(* POU FB_BACnet_RemoteAccumulator_EX, ST *)
FUNCTION_BLOCK FB_BACnet_RemoteAccumulator_EX
VAR_IN_OUT
	RemoteDevice		: FB_BACnet_RemoteDevice;
END_VAR
VAR_OUTPUT
	bReady				: BOOL;
	nPresentValue		: UDINT;
	bOverridden			: BOOL;
	bOutOfService		: BOOL;
	bFault				: BOOL;
	bInAlarm			: BOOL;
	bOverRange			: BOOL;
	bUnderRange			: BOOL;
	bNoSensor			: BOOL;
	bOpenLoop			: BOOL;
	bCommFailure		: BOOL;
	bShortedLoop		: BOOL;
	bOtherFault			: BOOL;
	tObjectID			: T_BACnet_ObjectIdentifier := 16#FFFFFFFF;
	bError				: BOOL;
	nErrorId			: UINT;
END_VAR
VAR
	_PresentValue AT%I*:UDINT;			(* ~(BACnet_PresentValue				:		: )
											(BACnet_ObjectType					: ACC	: )
											(BACnet_RemoteCycletimeRead			: 1000	: )
											(BACnet_RemoteFlagsRead				: 1		: )
											(BACnet_RemoteResubscriptionInterval: 240	: )
                                			(BACnet_RemoteCycleTimeWrite   		: 1000	: )
                                			(BACnet_RemoteFlagsWrite       		: 1		: )	*)
	_ObjectId AT%I*: DWORD;				(* ~(BACnet_ObjectIdentifier			:		: LINK) *)
	_StatusFlags AT%I*:WORD;			(* ~(BACnet_StatusFlags					:		: )	*)
	_Reliability AT%I*:WORD;			(* ~(BACnet_Reliability					:		: )	*)
	_StatusFlagsBits : ST_BACnet_StatusFlags;

	_nUpdateCount : UDINT := 0;
END_VAR
(* update client device *)
IF RemoteDevice._nUpdateCount = _nUpdateCount THEN
	RemoteDevice();
END_IF
(* remind current number of update counter *)
_nUpdateCount := RemoteDevice._nUpdateCount;

IF NOT RemoteDevice.bOperational THEN
	nErrorId := BACnet_ERR_OPERATIONAL;
	bReady := FALSE;

ELSIF (F_BACnet_GetObjType(_ObjectId) <> BACnetObjectType_Accumulator) THEN
	(* wrong mapping / invalid object ID *)
	IF _ObjectId = 0 THEN
		nErrorId := BACnet_ERR_WRONG_MAPPING;
	ELSE
		nErrorId := BACnet_ERR_INVALID_OBJECTID;
	END_IF
	bReady := FALSE;
	tObjectID := 16#FFFFFFFF;

ELSIF _StatusFlags >= 4 THEN
	(* clear error flag *)
	nErrorId := BACnet_ERR_NO_ERROR;
	bReady := TRUE;
	(* copy present value *)
	nPresentValue := _PresentValue;

	(* build bit states *)
	_StatusFlagsBits := F_BACnet_StatusFlags(_StatusFlags);

	(* copy states to output *)
	bOverridden := _StatusFlagsBits.overridden;
	bOutOfService := _StatusFlagsBits.out_of_service;
	bFault := _StatusFlagsBits.fault;
	bInAlarm := _StatusFlagsBits.in_alarm;
	bOverRange := (_Reliability = BACnetReliability_over_range);
	bUnderRange := (_Reliability = BACnetReliability_under_range);
	bNoSensor := (_Reliability = BACnetReliability_no_sensor);
	bOpenLoop := (_Reliability = BACnetReliability_open_loop);
	bCommFailure := (_Reliability = BACnetReliability_communication_failure);
	bShortedLoop := (_Reliability = BACnetReliability_shorted_loop);
	bOtherFault := (_Reliability = BACnetReliability_unreliable_other);
	tObjectID := _ObjectId;

ELSE
	bReady := FALSE;
	(* and set error ID *)
	nErrorId := BACnet_ERR_WRONG_MAPPING;
END_IF

(* set error flag *)
bError := (nErrorId <> BACnet_ERR_NO_ERROR);
END_FUNCTION_BLOCK

(* POU FB_BACnet_RemoteAnalogInput, ST *)
FUNCTION_BLOCK FB_BACnet_RemoteAnalogInput
VAR_IN_OUT
	RemoteDevice			: FB_BACnet_RemoteDevice;
END_VAR
VAR_OUTPUT
	bReady				: BOOL;
	fPresentValue		: REAL;
	bOverridden			: BOOL;
	bOutOfService		: BOOL;
	bFault				: BOOL;
	bInAlarm			: BOOL;
	bError				: BOOL;
	nErrorId			: UINT;
END_VAR
VAR
	_PresentValue AT%I*: REAL; 			(* ~(BACnet_PresentValue 				:		: )
								   			(BACnet_ObjectType 					: AI	: )
											(BACnet_RemoteCycletimeRead 		: 1000	: )
											(BACnet_RemoteFlagsRead        		: 1		: )
											(BACnet_RemoteResubscriptionInterval: 240	: )
	                                		(BACnet_RemoteCycleTimeWrite   		: 1000	: )
	                                		(BACnet_RemoteFlagsWrite       		: 1		: )	*)
	_StatusFlags AT%I*: WORD; 			(* ~(BACnet_StatusFlags 				:		: )	*)
	_StatusFlagsBits : ST_BACnet_StatusFlags;

	_nUpdateCount : UDINT := 0;
END_VAR
(* update client device *)
IF RemoteDevice._nUpdateCount = _nUpdateCount THEN
	RemoteDevice();
END_IF
(* remind current number of update counter *)
_nUpdateCount := RemoteDevice._nUpdateCount;

IF NOT RemoteDevice.bOperational THEN
	nErrorId := BACnet_ERR_OPERATIONAL;
	bReady := FALSE;

ELSIF _StatusFlags >= 4 THEN
	(* clear error flag *)
	nErrorId := BACnet_ERR_NO_ERROR;
	(* ready state *)
	bReady := TRUE;

	(* present value *)
	fPresentValue := _PresentValue;

	(* build bit states *)
	_StatusFlagsBits := F_BACnet_StatusFlags(_StatusFlags);

	(* copy states to output *)
	bOverridden := _StatusFlagsBits.overridden;
	bOutOfService := _StatusFlagsBits.out_of_service;
	bFault := _StatusFlagsBits.fault;
	bInAlarm := _StatusFlagsBits.in_alarm;
ELSE
	(* server device not ready, reset local ready also *)
	bReady := FALSE;
	(* and set error ID *)
	nErrorId := BACnet_ERR_WRONG_MAPPING;
END_IF

(* set error flag *)
bError := (nErrorId <> BACnet_ERR_NO_ERROR);
END_FUNCTION_BLOCK

(* POU FB_BACnet_RemoteAnalogInput_EX, ST *)
FUNCTION_BLOCK FB_BACnet_RemoteAnalogInput_EX
VAR_IN_OUT
	RemoteDevice			: FB_BACnet_RemoteDevice;
END_VAR
VAR_OUTPUT
	bReady				: BOOL;
	fPresentValue		: REAL;
	bOverridden			: BOOL;
	bOutOfService		: BOOL;
	bFault				: BOOL;
	bInAlarm			: BOOL;
	bOverRange			: BOOL;
	bUnderRange			: BOOL;
	bNoSensor			: BOOL;
	bOpenLoop			: BOOL;
	bShortedLoop		: BOOL;
	bOtherFault			: BOOL;
	eEventState			: E_BACNETEVENTSTATE;
	tObjectID			: T_BACnet_ObjectIdentifier := 16#FFFFFFFF;
	bError				: BOOL;
	nErrorId			: UINT;
END_VAR
VAR
	_PresentValue AT%I*: REAL; 			(* ~(BACnet_PresentValue 				:		: )
								   			(BACnet_ObjectType 					: AI	: )
											(BACnet_RemoteCycletimeRead 		: 1000	: )
											(BACnet_RemoteFlagsRead        		: 1		: )
											(BACnet_RemoteResubscriptionInterval: 240	: )
	                                		(BACnet_RemoteCycleTimeWrite   		: 1000	: )
	                                		(BACnet_RemoteFlagsWrite       		: 1		: )	*)
	_ObjectId AT%I*: DWORD;				(* ~(BACnet_ObjectIdentifier			:		: LINK) *)
	_StatusFlags AT%I*: WORD; 			(* ~(BACnet_StatusFlags 				:		: )	*)
	_Reliability AT%I*: WORD; 			(* ~(BACnet_Reliability 				:		: )	*)
	_EventState AT%I*: WORD;			(* ~(BACnet_EventState					:		: )	*)
	_nUpdateCount : UDINT := 0;
	_StatusFlagsBits : ST_BACnet_StatusFlags;
END_VAR
(* update client device *)
IF RemoteDevice._nUpdateCount = _nUpdateCount THEN
	RemoteDevice();
END_IF
(* remind current number of update counter *)
_nUpdateCount := RemoteDevice._nUpdateCount;

IF NOT RemoteDevice.bOperational THEN
	nErrorId := BACnet_ERR_OPERATIONAL;
	bReady := FALSE;

ELSIF (F_BACnet_GetObjType(_ObjectId) <> BACnetObjectType_AnalogInput) THEN
	(* wrong mapping / invalid object ID *)
	IF _ObjectId = 0 THEN
		nErrorId := BACnet_ERR_WRONG_MAPPING;
	ELSE
		nErrorId := BACnet_ERR_INVALID_OBJECTID;
	END_IF
	bReady := FALSE;
	tObjectID := 16#FFFFFFFF;

ELSIF _StatusFlags >= 4 THEN
	(* clear error flag *)
	nErrorId := BACnet_ERR_NO_ERROR;
	(* ready state *)
	bReady := TRUE;

	(* present value *)
	fPresentValue := _PresentValue;

	(* build bit states *)
	_StatusFlagsBits := F_BACnet_StatusFlags(_StatusFlags);

	(* copy states to output *)
	bOverridden := _StatusFlagsBits.overridden;
	bOutOfService := _StatusFlagsBits.out_of_service;
	bFault := _StatusFlagsBits.fault;
	bInAlarm := _StatusFlagsBits.in_alarm;
	bOverRange := (_Reliability = BACnetReliability_over_range);
	bUnderRange := (_Reliability = BACnetReliability_under_range);
	bNoSensor := (_Reliability = BACnetReliability_no_sensor);
	bOpenLoop := (_Reliability = BACnetReliability_open_loop);
	bShortedLoop := (_Reliability = BACnetReliability_shorted_loop);
	bOtherFault := (_Reliability = BACnetReliability_unreliable_other);
	eEventState := _EventState;
	tObjectID := _ObjectId;
ELSE
	(* server device not ready, reset local ready also *)
	bReady := FALSE;
	(* and set error ID *)
	nErrorId := BACnet_ERR_WRONG_MAPPING;
END_IF

(* set error flag *)
bError := (nErrorId <> BACnet_ERR_NO_ERROR);
END_FUNCTION_BLOCK

(* POU FB_BACnet_RemoteAnalogOutput, ST *)
FUNCTION_BLOCK FB_BACnet_RemoteAnalogOutput
VAR_IN_OUT
	RemoteDevice		: FB_BACnet_RemoteDevice;
END_VAR
VAR_OUTPUT
	bReady				: BOOL;
	fPresentValue		: REAL;
	bOverridden			: BOOL;
	bOutOfService		: BOOL;
	bFault				: BOOL;
	bInAlarm			: BOOL;
	bError				: BOOL;
	nErrorId			: UINT;
END_VAR
VAR
	_PresentValue AT%I*: REAL; 			(* ~(BACnet_PresentValue 				:		: )
								   			(BACnet_ObjectType 					: AO	: )
											(BACnet_RemoteCycletimeRead 		: 1000	: )
											(BACnet_RemoteFlagsRead        		: 1		: )
											(BACnet_RemoteResubscriptionInterval: 240	: )
	                                		(BACnet_RemoteCycleTimeWrite   		: 1000	: )
	                                		(BACnet_RemoteFlagsWrite       		: 1		: )	*)
	_StatusFlags AT%I*: WORD; 			(* ~(BACnet_StatusFlags 				:		: )	*)
	_StatusFlagsBits : ST_BACnet_StatusFlags;

	_nUpdateCount : UDINT := 0;
END_VAR
(* update client device *)
IF RemoteDevice._nUpdateCount = _nUpdateCount THEN
	RemoteDevice();
END_IF
(* remind current number of update counter *)
_nUpdateCount := RemoteDevice._nUpdateCount;

IF RemoteDevice.bFirstCycle THEN
	(* first call of the server device since reboot/reset *)
	bReady := FALSE;

ELSIF NOT RemoteDevice.bOperational THEN
	nErrorId := BACnet_ERR_OPERATIONAL;
	bReady := FALSE;

ELSIF _StatusFlags >= 4 THEN
	(* clear error flag *)
	nErrorId := BACnet_ERR_NO_ERROR;
	(* ready state *)
	bReady := TRUE;

	(* present value *)
	fPresentValue := _PresentValue;

	(* build bit states *)
	_StatusFlagsBits := F_BACnet_StatusFlags(_StatusFlags);

	(* copy states to output *)
	bOverridden := _StatusFlagsBits.overridden;
	bOutOfService := _StatusFlagsBits.out_of_service;
	bFault := _StatusFlagsBits.fault;
	bInAlarm := _StatusFlagsBits.in_alarm;
ELSE
	(* server device not ready, reset local ready also *)
	bReady := FALSE;
	(* and set error ID *)
	nErrorId := BACnet_ERR_WRONG_MAPPING;
END_IF

(* set error flag *)
bError := (nErrorId <> BACnet_ERR_NO_ERROR);
END_FUNCTION_BLOCK

(* POU FB_BACnet_RemoteAnalogOutput_EX, ST *)
FUNCTION_BLOCK FB_BACnet_RemoteAnalogOutput_EX
VAR_INPUT
	bEnablePV			: BOOL; (* enable present value with priority x in priority array, FALSE = priority x disable *)
	bNullPV				: BOOL; (* clear priority entry *)
	fPV					: REAL; (* decimal number for priority x, when input bEnablePV is TRUE *)
END_VAR
VAR_IN_OUT
	RemoteDevice		: FB_BACnet_RemoteDevice;
END_VAR
VAR_OUTPUT
	bReady				: BOOL;
	fPresentValue		: REAL;
	bOverridden			: BOOL;
	bOutOfService		: BOOL;
	bFault				: BOOL;
	bInAlarm			: BOOL;
	bNoOutput			: BOOL;
	bOpenLoop			: BOOL;
	bShortedLoop		: BOOL;
	bOtherFault			: BOOL;
	eEventState			: E_BACNETEVENTSTATE;
	tObjectID			: T_BACnet_ObjectIdentifier := 16#FFFFFFFF;
	bError				: BOOL;
	nErrorId			: UINT;
END_VAR
VAR
	_PresentValue AT%I*: REAL; 			(* ~(BACnet_PresentValue 				:		: )
								   			(BACnet_ObjectType 					: AO	: )
											(BACnet_RemoteCycletimeRead 		: 1000	: )
											(BACnet_RemoteFlagsRead        		: 1		: )
											(BACnet_RemoteResubscriptionInterval: 240	: )
	                                		(BACnet_RemoteCycleTimeWrite   		: 1000	: )
	                                		(BACnet_RemoteFlagsWrite       		: 1		: )	*)
    _PresentValue_Priority12 AT%Q*: DWORD;(* ~(BACnet_PresentValue_Priority12	:		: )	*)
	_ObjectId AT%I*: DWORD;				(* ~(BACnet_ObjectIdentifier			:		: LINK) *)
	_StatusFlags AT%I*: WORD; 			(* ~(BACnet_StatusFlags 				:		: )	*)
	_Reliability AT%I*: WORD; 			(* ~(BACnet_Reliability 				:		: )	*)
	_EventState AT%I*: WORD;			(* ~(BACnet_EventState					:		: )	*)
	_nUpdateCount : UDINT := 0;
	_StatusFlagsBits : ST_BACnet_StatusFlags;
END_VAR
(* update client device *)
IF RemoteDevice._nUpdateCount = _nUpdateCount THEN
	RemoteDevice();
END_IF
(* remind current number of update counter *)
_nUpdateCount := RemoteDevice._nUpdateCount;

IF RemoteDevice.bFirstCycle THEN
	(* first call of the server device since reboot/reset *)
	bReady := FALSE;
	_PresentValue_Priority12 := F_BACnet_RealNothing();

ELSIF NOT RemoteDevice.bOperational THEN
	nErrorId := BACnet_ERR_OPERATIONAL;
	bReady := FALSE;

ELSIF (F_BACnet_GetObjType(_ObjectId) <> BACnetObjectType_AnalogOutput) THEN
	(* wrong mapping / invalid object ID *)
	IF _ObjectId = 0 THEN
		nErrorId := BACnet_ERR_WRONG_MAPPING;
	ELSE
		nErrorId := BACnet_ERR_INVALID_OBJECTID;
	END_IF
	bReady := FALSE;
	tObjectID := 16#FFFFFFFF;

ELSIF _StatusFlags >= 4 THEN
	(* clear error flag *)
	nErrorId := BACnet_ERR_NO_ERROR;
	(* ready state *)
	bReady := TRUE;

	(* write into priority array *)
	_PresentValue_Priority12 := F_BACnet_RealPV(bEnablePV, bNullPV, fPV);

	(* present value *)
	fPresentValue := _PresentValue;

	(* build bit states *)
	_StatusFlagsBits := F_BACnet_StatusFlags(_StatusFlags);

	(* copy states to output *)
	bOverridden := _StatusFlagsBits.overridden;
	bOutOfService := _StatusFlagsBits.out_of_service;
	bFault := _StatusFlagsBits.fault;
	bInAlarm := _StatusFlagsBits.in_alarm;
	bNoOutput := (_Reliability = BACnetReliability_no_output);
	bOpenLoop := (_Reliability = BACnetReliability_open_loop);
	bShortedLoop := (_Reliability = BACnetReliability_shorted_loop);
	bOtherFault := (_Reliability = BACnetReliability_unreliable_other);
	eEventState := _EventState;
	tObjectID := _ObjectId;
ELSE
	(* server device not ready, reset local ready also *)
	bReady := FALSE;
	(* and set error ID *)
	nErrorId := BACnet_ERR_WRONG_MAPPING;
END_IF

(* set error flag *)
bError := (nErrorId <> BACnet_ERR_NO_ERROR);
END_FUNCTION_BLOCK

(* POU FB_BACnet_RemoteAnalogOutput_WR, ST *)
FUNCTION_BLOCK FB_BACnet_RemoteAnalogOutput_WR
VAR_INPUT
	bEnablePV			: BOOL; (* enable present value with priority x in priority array, FALSE = priority x disable *)
	bNullPV				: BOOL; (* clear priority entry *)
	fPV					: REAL; (* decimal number for priority x, when input bEnablePV is TRUE *)
END_VAR
VAR_IN_OUT
	RemoteDevice		: FB_BACnet_RemoteDevice;
END_VAR
VAR_OUTPUT
	bReady				: BOOL;
	fPresentValue		: REAL;
	bOverridden			: BOOL;
	bOutOfService		: BOOL;
	bFault				: BOOL;
	bInAlarm			: BOOL;
	bError				: BOOL;
	nErrorId			: UINT;
END_VAR
VAR
	_PresentValue AT%I*: REAL; 			(* ~(BACnet_PresentValue 				:		: )
								   			(BACnet_ObjectType 					: AO	: )
											(BACnet_RemoteCycletimeRead 		: 1000	: )
											(BACnet_RemoteFlagsRead        		: 1		: )
											(BACnet_RemoteResubscriptionInterval: 240	: )
	                                		(BACnet_RemoteCycleTimeWrite   		: 1000	: )
	                                		(BACnet_RemoteFlagsWrite       		: 1		: )	*)
    _PresentValue_Priority12 AT%Q*: DWORD;(* ~(BACnet_PresentValue_Priority12	:		: )	*)
	_StatusFlags AT%I*: WORD; 			(* ~(BACnet_StatusFlags 				:		: )	*)
	_StatusFlagsBits : ST_BACnet_StatusFlags;

	_nUpdateCount : UDINT := 0;
END_VAR
(* update client device *)
IF RemoteDevice._nUpdateCount = _nUpdateCount THEN
	RemoteDevice();
END_IF
(* remind current number of update counter *)
_nUpdateCount := RemoteDevice._nUpdateCount;

IF RemoteDevice.bFirstCycle THEN
	(* first call of the server device since reboot/reset *)
	bReady := FALSE;
	_PresentValue_Priority12 := F_BACnet_RealNothing();
ELSIF NOT RemoteDevice.bOperational THEN
	nErrorId := BACnet_ERR_OPERATIONAL;
	bReady := FALSE;

ELSIF _StatusFlags >= 4 THEN
	(* clear error flag *)
	nErrorId := BACnet_ERR_NO_ERROR;
	(* ready state *)
	bReady := TRUE;

	(* write into priority array *)
	_PresentValue_Priority12 := F_BACnet_RealPV(bEnablePV, bNullPV, fPV);

	(* present value *)
	fPresentValue := _PresentValue;

	(* build bit states *)
	_StatusFlagsBits := F_BACnet_StatusFlags(_StatusFlags);

	(* copy states to output *)
	bOverridden := _StatusFlagsBits.overridden;
	bOutOfService := _StatusFlagsBits.out_of_service;
	bFault := _StatusFlagsBits.fault;
	bInAlarm := _StatusFlagsBits.in_alarm;
ELSE
	(* server device not ready, reset local ready also *)
	bReady := FALSE;
	(* and set error ID *)
	nErrorId := BACnet_ERR_WRONG_MAPPING;
END_IF

(* set error flag *)
bError := (nErrorId <> BACnet_ERR_NO_ERROR);
END_FUNCTION_BLOCK

(* POU FB_BACnet_RemoteAnalogValue, ST *)
FUNCTION_BLOCK FB_BACnet_RemoteAnalogValue
VAR_IN_OUT
	RemoteDevice		: FB_BACnet_RemoteDevice;
END_VAR
VAR_OUTPUT
	bReady				: BOOL;
	fPresentValue		: REAL;
	bOverridden			: BOOL;
	bOutOfService		: BOOL;
	bFault				: BOOL;
	bInAlarm			: BOOL;
	bError				: BOOL;
	nErrorId			: UINT;
END_VAR
VAR
	_PresentValue AT%I*: REAL; 			(* ~(BACnet_PresentValue 				:		: )
								   			(BACnet_ObjectType 					: AV	: )
											(BACnet_RemoteCycletimeRead 		: 1000	: )
											(BACnet_RemoteFlagsRead        		: 1		: )
											(BACnet_RemoteResubscriptionInterval: 240	: )
	                                		(BACnet_RemoteCycleTimeWrite   		: 1000	: )
	                                		(BACnet_RemoteFlagsWrite       		: 1		: )	*)
	_StatusFlags AT%I*: WORD; 			(* ~(BACnet_StatusFlags 				:		: )	*)
	_StatusFlagsBits : ST_BACnet_StatusFlags;

	_nUpdateCount : UDINT := 0;
END_VAR
(* update client device *)
IF RemoteDevice._nUpdateCount = _nUpdateCount THEN
	RemoteDevice();
END_IF
(* remind current number of update counter *)
_nUpdateCount := RemoteDevice._nUpdateCount;

IF RemoteDevice.bFirstCycle THEN
	(* first call of the server device since reboot/reset *)
	bReady := FALSE;

ELSIF NOT RemoteDevice.bOperational THEN
	nErrorId := BACnet_ERR_OPERATIONAL;
	bReady := FALSE;

ELSIF _StatusFlags >= 4 THEN
	(* clear error flag *)
	nErrorId := BACnet_ERR_NO_ERROR;
	(* ready state *)
	bReady := TRUE;

	(* present value *)
	fPresentValue := _PresentValue;

	(* build bit states *)
	_StatusFlagsBits := F_BACnet_StatusFlags(_StatusFlags);

	(* copy states to output *)
	bOverridden := _StatusFlagsBits.overridden;
	bOutOfService := _StatusFlagsBits.out_of_service;
	bFault := _StatusFlagsBits.fault;
	bInAlarm := _StatusFlagsBits.in_alarm;
ELSE
	(* server device not ready, reset local ready also *)
	bReady := FALSE;
	(* and set error ID *)
	nErrorId := BACnet_ERR_WRONG_MAPPING;
END_IF

(* set error flag *)
bError := (nErrorId <> BACnet_ERR_NO_ERROR);
END_FUNCTION_BLOCK

(* POU FB_BACnet_RemoteAnalogValue_EX, ST *)
FUNCTION_BLOCK FB_BACnet_RemoteAnalogValue_EX
VAR_INPUT
	bEnablePV			: BOOL; (* enable present value with priority x in priority array, FALSE = priority x disable *)
	bNullPV				: BOOL; (* clear priority entry *)
	fPV					: REAL; (* decimal number for priority x, when input bEnablePV is TRUE *)
END_VAR
VAR_IN_OUT
	RemoteDevice		: FB_BACnet_RemoteDevice;
END_VAR
VAR_OUTPUT
	bReady				: BOOL;
	fPresentValue		: REAL;
	bOverridden			: BOOL;
	bOutOfService		: BOOL;
	bFault				: BOOL;
	bInAlarm			: BOOL;
	bOverRange			: BOOL;
	bUnderRange			: BOOL;
	bOtherFault			: BOOL;
	eEventState			: E_BACNETEVENTSTATE;
	tObjectID			: T_BACnet_ObjectIdentifier := 16#FFFFFFFF;
	bError				: BOOL;
	nErrorId			: UINT;
END_VAR
VAR
	_PresentValue AT%I*: REAL; 			(* ~(BACnet_PresentValue 				:		: )
								   			(BACnet_ObjectType 					: AV	: )
											(BACnet_RemoteCycletimeRead 		: 1000	: )
											(BACnet_RemoteFlagsRead        		: 1		: )
											(BACnet_RemoteResubscriptionInterval: 240	: )
	                                		(BACnet_RemoteCycleTimeWrite   		: 1000	: )
	                                		(BACnet_RemoteFlagsWrite       		: 1		: )	*)
    _PresentValue_Priority12 AT%Q*: DWORD;(* ~(BACnet_PresentValue_Priority12	:		: )	*)
	_ObjectId AT%I*: DWORD;				(* ~(BACnet_ObjectIdentifier			:		: LINK) *)
	_StatusFlags AT%I*: WORD; 			(* ~(BACnet_StatusFlags 				:		: )	*)
	_Reliability AT%I*: WORD;			(* ~(BACnet_Reliability 				:		: )	*)
	_EventState AT%I*: WORD;			(* ~(BACnet_EventState					:		: )	*)
	_nUpdateCount : UDINT := 0;
	_StatusFlagsBits : ST_BACnet_StatusFlags;
END_VAR
(* update client device *)
IF RemoteDevice._nUpdateCount = _nUpdateCount THEN
	RemoteDevice();
END_IF
(* remind current number of update counter *)
_nUpdateCount := RemoteDevice._nUpdateCount;

IF RemoteDevice.bFirstCycle THEN
	(* first call of the server device since reboot/reset *)
	bReady := FALSE;
	_PresentValue_Priority12 := F_BACnet_RealNothing();
ELSIF NOT RemoteDevice.bOperational THEN
	nErrorId := BACnet_ERR_OPERATIONAL;
	bReady := FALSE;

ELSIF (F_BACnet_GetObjType(_ObjectId) <> BACnetObjectType_AnalogValue) THEN
	(* wrong mapping / invalid object ID *)
	IF _ObjectId = 0 THEN
		nErrorId := BACnet_ERR_WRONG_MAPPING;
	ELSE
		nErrorId := BACnet_ERR_INVALID_OBJECTID;
	END_IF
	bReady := FALSE;
	tObjectID := 16#FFFFFFFF;

ELSIF _StatusFlags >= 4 THEN
	(* clear error flag *)
	nErrorId := BACnet_ERR_NO_ERROR;
	(* ready state *)
	bReady := TRUE;

	(* write into priority array *)
	_PresentValue_Priority12 := F_BACnet_RealPV(bEnablePV, bNullPV, fPV);

	(* present value *)
	fPresentValue := _PresentValue;

	(* build bit states *)
	_StatusFlagsBits := F_BACnet_StatusFlags(_StatusFlags);

	(* copy states to output *)
	bOverridden := _StatusFlagsBits.overridden;
	bOutOfService := _StatusFlagsBits.out_of_service;
	bFault := _StatusFlagsBits.fault;
	bInAlarm := _StatusFlagsBits.in_alarm;
	bOverRange := (_Reliability = BACnetReliability_over_range);
	bUnderRange := (_Reliability = BACnetReliability_under_range);
	bOtherFault := (_Reliability = BACnetReliability_unreliable_other);
	eEventState := _EventState;
	tObjectID := _ObjectId;
ELSE
	(* server device not ready, reset local ready also *)
	bReady := FALSE;
	(* and set error ID *)
	nErrorId := BACnet_ERR_WRONG_MAPPING;
END_IF

(* set error flag *)
bError := (nErrorId <> BACnet_ERR_NO_ERROR);
END_FUNCTION_BLOCK

(* POU FB_BACnet_RemoteAnalogValue_WR, ST *)
FUNCTION_BLOCK FB_BACnet_RemoteAnalogValue_WR
VAR_INPUT
	bEnablePV			: BOOL; (* enable present value with priority x in priority array, FALSE = priority x disable *)
	bNullPV				: BOOL; (* clear priority entry *)
	fPV					: REAL; (* decimal number for priority x, when input bEnablePV is TRUE *)
END_VAR
VAR_IN_OUT
	RemoteDevice		: FB_BACnet_RemoteDevice;
END_VAR
VAR_OUTPUT
	bReady				: BOOL;
	fPresentValue		: REAL;
	bOverridden			: BOOL;
	bOutOfService		: BOOL;
	bFault				: BOOL;
	bInAlarm			: BOOL;
	bError				: BOOL;
	nErrorId			: UINT;
END_VAR
VAR
	_PresentValue AT%I*: REAL; 			(* ~(BACnet_PresentValue 				:		: )
								   			(BACnet_ObjectType 					: AV	: )
											(BACnet_RemoteCycletimeRead 		: 1000	: )
											(BACnet_RemoteFlagsRead        		: 1		: )
											(BACnet_RemoteResubscriptionInterval: 240	: )
	                                		(BACnet_RemoteCycleTimeWrite   		: 1000	: )
	                                		(BACnet_RemoteFlagsWrite       		: 1		: )	*)
    _PresentValue_Priority12 AT%Q*: DWORD;(* ~(BACnet_PresentValue_Priority12	:		: )	*)
	_StatusFlags AT%I*: WORD; 			(* ~(BACnet_StatusFlags 				:		: )	*)
	_StatusFlagsBits : ST_BACnet_StatusFlags;

	_nUpdateCount : UDINT := 0;
END_VAR
(* update client device *)
IF RemoteDevice._nUpdateCount = _nUpdateCount THEN
	RemoteDevice();
END_IF
(* remind current number of update counter *)
_nUpdateCount := RemoteDevice._nUpdateCount;

IF RemoteDevice.bFirstCycle THEN
	(* first call of the server device since reboot/reset *)
	bReady := FALSE;
	_PresentValue_Priority12 := F_BACnet_RealNothing();
ELSIF NOT RemoteDevice.bOperational THEN
	nErrorId := BACnet_ERR_OPERATIONAL;
	bReady := FALSE;

ELSIF _StatusFlags >= 4 THEN
	(* clear error flag *)
	nErrorId := BACnet_ERR_NO_ERROR;
	(* ready state *)
	bReady := TRUE;

	(* write into priority array *)
	_PresentValue_Priority12 := F_BACnet_RealPV(bEnablePV, bNullPV, fPV);

	(* present value *)
	fPresentValue := _PresentValue;

	(* build bit states *)
	_StatusFlagsBits := F_BACnet_StatusFlags(_StatusFlags);

	(* copy states to output *)
	bOverridden := _StatusFlagsBits.overridden;
	bOutOfService := _StatusFlagsBits.out_of_service;
	bFault := _StatusFlagsBits.fault;
	bInAlarm := _StatusFlagsBits.in_alarm;
ELSE
	(* server device not ready, reset local ready also *)
	bReady := FALSE;
	(* and set error ID *)
	nErrorId := BACnet_ERR_WRONG_MAPPING;
END_IF

(* set error flag *)
bError := (nErrorId <> BACnet_ERR_NO_ERROR);
END_FUNCTION_BLOCK

(* POU FB_BACnet_RemoteAveraging, ST *)
FUNCTION_BLOCK FB_BACnet_RemoteAveraging
VAR_IN_OUT
	RemoteDevice		: FB_BACnet_RemoteDevice;
END_VAR
VAR_OUTPUT
	bReady				: BOOL;
	nAverageValue		: REAL;
	bError				: BOOL;
	nErrorId			: UINT;
END_VAR
VAR
	_AverageValue AT%I*: REAL; 		(* ~(BACnet_AverageValue 				:		: )
										(BACnet_ObjectType					: AVG  	: )
										(BACnet_RemoteCycletimeRead 		: 1000	: )
										(BACnet_RemoteFlagsRead        		: 1		: )
										(BACnet_RemoteResubscriptionInterval: 240	: )
										(BACnet_RemoteCycleTimeWrite   		: 1000	: )
										(BACnet_RemoteFlagsWrite       		: 1		: )	*)

	_nUpdateCount : UDINT := 0;
END_VAR
(* update client device *)
IF RemoteDevice._nUpdateCount = _nUpdateCount THEN
	RemoteDevice();
END_IF
(* remind current number of update counter *)
_nUpdateCount := RemoteDevice._nUpdateCount;

IF RemoteDevice.bOperational THEN
	(* clear error flag *)
	nErrorId := BACnet_ERR_NO_ERROR;
	(* ready state *)
	bReady := TRUE;
	(* present value *)
	nAverageValue := _AverageValue;
ELSE
	(* server device not ready, reset local ready also *)
	bReady := FALSE;
	(* and set error ID *)
	nErrorId := BACnet_ERR_OPERATIONAL;
END_IF

(* set error flag *)
bError := (nErrorId <> BACnet_ERR_NO_ERROR);
END_FUNCTION_BLOCK

(* POU FB_BACnet_RemoteAveraging_EX, ST *)
FUNCTION_BLOCK FB_BACnet_RemoteAveraging_EX
VAR_IN_OUT
	RemoteDevice		: FB_BACnet_RemoteDevice;
END_VAR
VAR_OUTPUT
	bReady				: BOOL;
	nAverageValue		: REAL;
	tObjectID			: T_BACnet_ObjectIdentifier := 16#FFFFFFFF;
	bError				: BOOL;
	nErrorId			: UINT;
END_VAR
VAR
	_AverageValue AT%I*: REAL; 		(* ~(BACnet_AverageValue 				:		: )
										(BACnet_ObjectType					: AVG  	: )
										(BACnet_RemoteCycletimeRead 		: 1000	: )
										(BACnet_RemoteFlagsRead        		: 1		: )
										(BACnet_RemoteResubscriptionInterval: 240	: )
										(BACnet_RemoteCycleTimeWrite   		: 1000	: )
										(BACnet_RemoteFlagsWrite       		: 1		: )	*)
	_ObjectId AT%I*: DWORD;			(* ~(BACnet_ObjectIdentifier			:		: LINK) *)

	_nUpdateCount : UDINT := 0;
END_VAR
(* update client device *)
IF RemoteDevice._nUpdateCount = _nUpdateCount THEN
	RemoteDevice();
END_IF
(* remind current number of update counter *)
_nUpdateCount := RemoteDevice._nUpdateCount;

IF NOT RemoteDevice.bOperational THEN
	(* server device not ready, reset local ready also *)
	bReady := FALSE;
	(* and set error ID *)
	nErrorId := BACnet_ERR_OPERATIONAL;

ELSIF (F_BACnet_GetObjType(_ObjectId) <> BACnetObjectType_Averaging) THEN
	(* wrong mapping / invalid object ID *)
	IF _ObjectId = 0 THEN
		nErrorId := BACnet_ERR_WRONG_MAPPING;
	ELSE
		nErrorId := BACnet_ERR_INVALID_OBJECTID;
	END_IF
	bReady := FALSE;
	tObjectID := 16#FFFFFFFF;

ELSE
	(* clear error flag *)
	nErrorId := BACnet_ERR_NO_ERROR;
	(* ready state *)
	bReady := TRUE;
	(* present value *)
	nAverageValue := _AverageValue;
	tObjectID := _ObjectId;

END_IF

(* set error flag *)
bError := (nErrorId <> BACnet_ERR_NO_ERROR);
END_FUNCTION_BLOCK

(* POU FB_BACnet_RemoteBinaryInput, ST *)
FUNCTION_BLOCK FB_BACnet_RemoteBinaryInput
VAR_OUTPUT
	bReady				: BOOL;
	bPresentValue		: BOOL;
	bOverridden			: BOOL;
	bOutOfService		: BOOL;
	bFault				: BOOL;
	bInAlarm			: BOOL;
	bError				: BOOL;
	nErrorId			: UINT;
END_VAR
VAR_IN_OUT
	RemoteDevice			: FB_BACnet_RemoteDevice;
END_VAR
VAR
	_PresentValue AT%I*: WORD; 				(* ~(BACnet_PresentValue 				:		: )
												(BACnet_ObjectType					: BI    : )
												(BACnet_RemoteCycletimeRead 		: 1000	: )
												(BACnet_RemoteFlagsRead        		: 1		: )
												(BACnet_RemoteResubscriptionInterval: 240	: )
		                                		(BACnet_RemoteCycleTimeWrite   		: 1000	: )
		                                		(BACnet_RemoteFlagsWrite       		: 1		: )	*)
	_StatusFlags AT%I*: WORD; 				(* ~(BACnet_StatusFlags 				:	    : )	*)
	_StatusFlagsBits : ST_BACnet_StatusFlags;
	_nUpdateCount : UDINT := 0;
END_VAR
(* update client device *)
IF RemoteDevice._nUpdateCount = _nUpdateCount THEN
	RemoteDevice();
END_IF
(* remind current number of update counter *)
_nUpdateCount := RemoteDevice._nUpdateCount;

IF NOT RemoteDevice.bOperational THEN
	nErrorId := BACnet_ERR_OPERATIONAL;
	bReady := FALSE;

ELSIF _StatusFlags >= 4 THEN
	(* clear error flag *)
	nErrorId := BACnet_ERR_NO_ERROR;
	(* ready state *)
	bReady := TRUE;

	(* present value *)
	bPresentValue := F_BinPV_To_Bool(_PresentValue);

	(* build bit states *)
	_StatusFlagsBits := F_BACnet_StatusFlags(_StatusFlags);

	(* copy states to output *)
	bOverridden := _StatusFlagsBits.overridden;
	bOutOfService := _StatusFlagsBits.out_of_service;
	bFault := _StatusFlagsBits.fault;
	bInAlarm := _StatusFlagsBits.in_alarm;

ELSE
	bReady := FALSE;
	(* and set error ID *)
	nErrorId := BACnet_ERR_WRONG_MAPPING;
END_IF

(* set error flag *)
bError := (nErrorId <> BACnet_ERR_NO_ERROR);
END_FUNCTION_BLOCK

(* POU FB_BACnet_RemoteBinaryInput_EX, ST *)
FUNCTION_BLOCK FB_BACnet_RemoteBinaryInput_EX
VAR_OUTPUT
	bReady				: BOOL;
	bPresentValue		: BOOL;
	bOverridden			: BOOL;
	bOutOfService		: BOOL;
	bFault				: BOOL;
	bInAlarm			: BOOL;
	bNoSensor			: BOOL;
	bOpenLoop			: BOOL;
	bShortedLoop		: BOOL;
	bOtherFault			: BOOL;
	eEventState			: E_BACNETEVENTSTATE;
	nChangeOfState		: UDINT;
	tObjectID			: T_BACnet_ObjectIdentifier := 16#FFFFFFFF;
	bError				: BOOL;
	nErrorId			: UINT;
END_VAR
VAR_IN_OUT
	RemoteDevice			: FB_BACnet_RemoteDevice;
END_VAR
VAR
	_ChangeOfStateCount AT%I*: UDINT;	(* ~(BACnet_ChangeOfStateCount			:		: ) *)
	_ObjectId AT%I*: DWORD;				(* ~(BACnet_ObjectIdentifier			:		: LINK) *)
	_PresentValue AT%I*: WORD; 			(* ~(BACnet_PresentValue 				:		: )
											(BACnet_ObjectType					: BI    : )
											(BACnet_RemoteCycletimeRead 		: 1000	: )
											(BACnet_RemoteFlagsRead        		: 1		: )
											(BACnet_RemoteResubscriptionInterval: 240	: )
		                                	(BACnet_RemoteCycleTimeWrite   		: 1000	: )
		                                	(BACnet_RemoteFlagsWrite       		: 1		: )	*)
	_StatusFlags AT%I*: WORD; 			(* ~(BACnet_StatusFlags 				:	    : )	*)
	_Reliability AT%I*: WORD; 			(* ~(BACnet_Reliability 				:		: )	*)
	_EventState AT%I*: WORD;			(* ~(BACnet_EventState					:		: )	*)
	_nUpdateCount : UDINT := 0;
	_StatusFlagsBits : ST_BACnet_StatusFlags;
END_VAR
(* update client device *)
IF RemoteDevice._nUpdateCount = _nUpdateCount THEN
	RemoteDevice();
END_IF
(* remind current number of update counter *)
_nUpdateCount := RemoteDevice._nUpdateCount;

IF NOT RemoteDevice.bOperational THEN
	nErrorId := BACnet_ERR_OPERATIONAL;
	bReady := FALSE;

ELSIF (F_BACnet_GetObjType(_ObjectId) <> BACnetObjectType_BinaryInput) THEN
	(* wrong mapping / invalid object ID *)
	IF _ObjectId = 0 THEN
		nErrorId := BACnet_ERR_WRONG_MAPPING;
	ELSE
		nErrorId := BACnet_ERR_INVALID_OBJECTID;
	END_IF
	bReady := FALSE;
	tObjectID := 16#FFFFFFFF;

ELSIF _StatusFlags >= 4 THEN
	(* clear error flag *)
	nErrorId := BACnet_ERR_NO_ERROR;
	(* ready state *)
	bReady := TRUE;

	(* present value *)
	bPresentValue := F_BinPV_To_Bool(_PresentValue);

	(* build bit states *)
	_StatusFlagsBits := F_BACnet_StatusFlags(_StatusFlags);

	(* copy states to output *)
	bOverridden := _StatusFlagsBits.overridden;
	bOutOfService := _StatusFlagsBits.out_of_service;
	bFault := _StatusFlagsBits.fault;
	bInAlarm := _StatusFlagsBits.in_alarm;
	bNoSensor := (_Reliability = BACnetReliability_no_sensor);
	bOpenLoop := (_Reliability = BACnetReliability_open_loop);
	bShortedLoop := (_Reliability = BACnetReliability_shorted_loop);
	bOtherFault := (_Reliability = BACnetReliability_unreliable_other);
	eEventState := _EventState;
	tObjectID := _ObjectId;

	(* copy change_of_state_count *)
	nChangeOfState := _ChangeOfStateCount;

ELSE
	bReady := FALSE;
	(* and set error ID *)
	nErrorId := BACnet_ERR_WRONG_MAPPING;
END_IF

(* set error flag *)
bError := (nErrorId <> BACnet_ERR_NO_ERROR);
END_FUNCTION_BLOCK

(* POU FB_BACnet_RemoteBinaryOutput, ST *)
FUNCTION_BLOCK FB_BACnet_RemoteBinaryOutput
VAR_IN_OUT
	RemoteDevice		: FB_BACnet_RemoteDevice;
END_VAR
VAR_OUTPUT
	bReady				: BOOL;
	bPresentValue		: BOOL;
	bOverridden			: BOOL;
	bOutOfService		: BOOL;
	bFault				: BOOL;
	bInAlarm			: BOOL;
	bError				: BOOL;
	nErrorId			: UINT;
END_VAR
VAR
	_PresentValue AT%I*: WORD; 			(* ~(BACnet_PresentValue 				:		: )
								   			(BACnet_ObjectType 					: BO	: )
											(BACnet_RemoteCycletimeRead 		: 1000	: )
											(BACnet_RemoteFlagsRead        		: 1		: )
											(BACnet_RemoteResubscriptionInterval: 240	: )
		                            		(BACnet_RemoteCycleTimeWrite   		: 1000	: )
		                            		(BACnet_RemoteFlagsWrite       		: 1		: )	*)
	_StatusFlags AT%I*: WORD; 			(* ~(BACnet_StatusFlags 				:		: )	*)
	_StatusFlagsBits : ST_BACnet_StatusFlags;
	_nUpdateCount : UDINT := 0;
END_VAR
(* update client device *)
IF RemoteDevice._nUpdateCount = _nUpdateCount THEN
	RemoteDevice();
END_IF
(* remind current number of update counter *)
_nUpdateCount := RemoteDevice._nUpdateCount;

IF RemoteDevice.bFirstCycle THEN
	(* first call of the server device since reboot/reset *)
	bReady := FALSE;

ELSIF NOT RemoteDevice.bOperational THEN
	nErrorId := BACnet_ERR_OPERATIONAL;
	bReady := FALSE;

ELSIF _StatusFlags >= 4 THEN
	(* clear error flag *)
	nErrorId := BACnet_ERR_NO_ERROR;
	(* ready state *)
	bReady := TRUE;

	(* present value *)
	bPresentValue := F_BinPV_To_Bool(_PresentValue);

	(* build bit states *)
	_StatusFlagsBits := F_BACnet_StatusFlags(_StatusFlags);

	(* copy states to output *)
	bOverridden := _StatusFlagsBits.overridden;
	bOutOfService := _StatusFlagsBits.out_of_service;
	bFault := _StatusFlagsBits.fault;
	bInAlarm := _StatusFlagsBits.in_alarm;
ELSE
	(* server device not ready, reset local ready also *)
	bReady := FALSE;
	(* and set error ID *)
	nErrorId := BACnet_ERR_WRONG_MAPPING;
END_IF

(* set error flag *)
bError := (nErrorId <> BACnet_ERR_NO_ERROR);
END_FUNCTION_BLOCK

(* POU FB_BACnet_RemoteBinaryOutput_EX, ST *)
FUNCTION_BLOCK FB_BACnet_RemoteBinaryOutput_EX
VAR_INPUT
	bEnablePV			: BOOL; (* enable present value with priority x in priority array, FALSE = priority x disable *)
	bNullPV				: BOOL; (* clear priority entry *)
	bPV					: BOOL; (* present value bool type *)
END_VAR
VAR_IN_OUT
	RemoteDevice		: FB_BACnet_RemoteDevice;
END_VAR
VAR_OUTPUT
	bReady				: BOOL;
	bPresentValue		: BOOL;
	bOverridden			: BOOL;
	bOutOfService		: BOOL;
	bFault				: BOOL;
	bInAlarm			: BOOL;
	bNoOutput			: BOOL;
	bOpenLoop			: BOOL;
	bShortedLoop		: BOOL;
	bOtherFault			: BOOL;
	eEventState			: E_BACNETEVENTSTATE;
	nChangeOfState		: UDINT;
	tObjectID			: T_BACnet_ObjectIdentifier := 16#FFFFFFFF;
	bError				: BOOL;
	nErrorId			: UINT;
END_VAR
VAR
	_ChangeOfStateCount AT%I*: UDINT;	(* ~(BACnet_ChangeOfStateCount			:		: ) *)
	_ObjectId AT%I*: DWORD;				(* ~(BACnet_ObjectIdentifier			:		: LINK) *)
	_PresentValue AT%I*: WORD; 			(* ~(BACnet_PresentValue 				:		: )
								   			(BACnet_ObjectType 					: BO	: )
											(BACnet_RemoteCycletimeRead 		: 1000	: )
											(BACnet_RemoteFlagsRead        		: 1		: )
											(BACnet_RemoteResubscriptionInterval: 240	: )
		                            		(BACnet_RemoteCycleTimeWrite   		: 1000	: )
		                            		(BACnet_RemoteFlagsWrite       		: 1		: )	*)
	_StatusFlags AT%I*: WORD; 			(* ~(BACnet_StatusFlags 				:		: )	*)
	_Reliability AT%I*: WORD;			(* ~(BACnet_Reliability 				:		: )	*)
	_EventState AT%I*: WORD;			(* ~(BACnet_EventState					:		: )	*)
    _PresentValue_Priority12 AT%Q*: WORD;(* ~(BACnet_PresentValue_Priority12	:		: )	*)
	_nUpdateCount : UDINT := 0;
	_StatusFlagsBits : ST_BACnet_StatusFlags;
END_VAR
(* update client device *)
IF RemoteDevice._nUpdateCount = _nUpdateCount THEN
	RemoteDevice();
END_IF
(* remind current number of update counter *)
_nUpdateCount := RemoteDevice._nUpdateCount;

IF RemoteDevice.bFirstCycle THEN
	(* first call of the server device since reboot/reset *)
	bReady := FALSE;
	_PresentValue_Priority12 := BACnetBinaryPV_Nothing;
ELSIF NOT RemoteDevice.bOperational THEN
	nErrorId := BACnet_ERR_OPERATIONAL;
	bReady := FALSE;

ELSIF (F_BACnet_GetObjType(_ObjectId) <> BACnetObjectType_BinaryOutput) THEN
	(* wrong mapping / invalid object ID *)
	IF _ObjectId = 0 THEN
		nErrorId := BACnet_ERR_WRONG_MAPPING;
	ELSE
		nErrorId := BACnet_ERR_INVALID_OBJECTID;
	END_IF
	bReady := FALSE;
	tObjectID := 16#FFFFFFFF;

ELSIF _StatusFlags >= 4 THEN
	(* clear error flag *)
	nErrorId := BACnet_ERR_NO_ERROR;
	(* ready state *)
	bReady := TRUE;

	(* write into priority array *)
	_PresentValue_Priority12 := F_Bool_To_BinPV(bEnablePV, bNullPV, bPV);

	(* present value *)
	bPresentValue := F_BinPV_To_Bool(_PresentValue);

	(* build bit states *)
	_StatusFlagsBits := F_BACnet_StatusFlags(_StatusFlags);

	(* copy states to output *)
	bOverridden := _StatusFlagsBits.overridden;
	bOutOfService := _StatusFlagsBits.out_of_service;
	bFault := _StatusFlagsBits.fault;
	bInAlarm := _StatusFlagsBits.in_alarm;
	bNoOutput := (_Reliability = BACnetReliability_no_output);
	bOpenLoop := (_Reliability = BACnetReliability_open_loop);
	bShortedLoop := (_Reliability = BACnetReliability_shorted_loop);
	bOtherFault := (_Reliability = BACnetReliability_unreliable_other);
	eEventState := _EventState;
	tObjectID := _ObjectId;

	(* copy change_of_state_count *)
	nChangeOfState := _ChangeOfStateCount;
ELSE
	(* server device not ready, reset local ready also *)
	bReady := FALSE;
	(* and set error ID *)
	nErrorId := BACnet_ERR_WRONG_MAPPING;
END_IF

(* set error flag *)
bError := (nErrorId <> BACnet_ERR_NO_ERROR);
END_FUNCTION_BLOCK

(* POU FB_BACnet_RemoteBinaryOutput_WR, ST *)
FUNCTION_BLOCK FB_BACnet_RemoteBinaryOutput_WR
VAR_INPUT
	bEnablePV			: BOOL; (* enable present value with priority x in priority array, FALSE = priority x disable *)
	bNullPV				: BOOL; (* clear priority entry *)
	bPV					: BOOL; (* present value bool type *)
END_VAR
VAR_IN_OUT
	RemoteDevice		: FB_BACnet_RemoteDevice;
END_VAR
VAR_OUTPUT
	bReady				: BOOL;
	bPresentValue		: BOOL;
	bOverridden			: BOOL;
	bOutOfService		: BOOL;
	bFault				: BOOL;
	bInAlarm			: BOOL;
	bError				: BOOL;
	nErrorId			: UINT;
END_VAR
VAR
	_PresentValue AT%I*: WORD; 			(* ~(BACnet_PresentValue 				:		: )
								   			(BACnet_ObjectType 					: BO	: )
											(BACnet_RemoteCycletimeRead 		: 1000	: )
											(BACnet_RemoteFlagsRead        		: 1		: )
											(BACnet_RemoteResubscriptionInterval: 240	: )
		                            		(BACnet_RemoteCycleTimeWrite   		: 1000	: )
		                            		(BACnet_RemoteFlagsWrite       		: 1		: )	*)
    _PresentValue_Priority12 AT%Q*: WORD;(* ~(BACnet_PresentValue_Priority12	:		: )	*)
	_StatusFlags AT%I*: WORD; 			(* ~(BACnet_StatusFlags 				:		: )	*)
	_StatusFlagsBits : ST_BACnet_StatusFlags;
	_nUpdateCount : UDINT := 0;
END_VAR
(* update client device *)
IF RemoteDevice._nUpdateCount = _nUpdateCount THEN
	RemoteDevice();
END_IF
(* remind current number of update counter *)
_nUpdateCount := RemoteDevice._nUpdateCount;

IF RemoteDevice.bFirstCycle THEN
	(* first call of the server device since reboot/reset *)
	bReady := FALSE;
	_PresentValue_Priority12 := BACnetBinaryPV_Nothing;
ELSIF NOT RemoteDevice.bOperational THEN
	nErrorId := BACnet_ERR_OPERATIONAL;
	bReady := FALSE;

ELSIF _StatusFlags >= 4 THEN
	(* clear error flag *)
	nErrorId := BACnet_ERR_NO_ERROR;
	(* ready state *)
	bReady := TRUE;

	(* write into priority array *)
	_PresentValue_Priority12 := F_Bool_To_BinPV(bEnablePV, bNullPV, bPV);

	(* present value *)
	bPresentValue := F_BinPV_To_Bool(_PresentValue);

	(* build bit states *)
	_StatusFlagsBits := F_BACnet_StatusFlags(_StatusFlags);

	(* copy states to output *)
	bOverridden := _StatusFlagsBits.overridden;
	bOutOfService := _StatusFlagsBits.out_of_service;
	bFault := _StatusFlagsBits.fault;
	bInAlarm := _StatusFlagsBits.in_alarm;
ELSE
	(* server device not ready, reset local ready also *)
	bReady := FALSE;
	(* and set error ID *)
	nErrorId := BACnet_ERR_WRONG_MAPPING;
END_IF

(* set error flag *)
bError := (nErrorId <> BACnet_ERR_NO_ERROR);
END_FUNCTION_BLOCK

(* POU FB_BACnet_RemoteBinaryValue, ST *)
FUNCTION_BLOCK FB_BACnet_RemoteBinaryValue
VAR_IN_OUT
	RemoteDevice		: FB_BACnet_RemoteDevice;
END_VAR
VAR_OUTPUT
	bReady				: BOOL;
	bPresentValue		: BOOL;
	bOverridden			: BOOL;
	bOutOfService		: BOOL;
	bFault				: BOOL;
	bInAlarm			: BOOL;
	bError				: BOOL;
	nErrorId			: UINT;
END_VAR
VAR

	_PresentValue AT%I*: WORD; 			(* ~(BACnet_PresentValue 				:		: )
								   			(BACnet_ObjectType 					: BV	: )
											(BACnet_RemoteCycletimeRead 		: 1000	: )
											(BACnet_RemoteFlagsRead        		: 1		: )
											(BACnet_RemoteResubscriptionInterval: 240	: )
	                                		(BACnet_RemoteCycleTimeWrite   		: 1000	: )
	                                		(BACnet_RemoteFlagsWrite       		: 1		: )	*)
	_StatusFlags AT%I*: WORD; 			(* ~(BACnet_StatusFlags 				:		: )	*)
	_StatusFlagsBits : ST_BACnet_StatusFlags;

	_nUpdateCount : UDINT := 0;
END_VAR
(* update client device *)
IF RemoteDevice._nUpdateCount = _nUpdateCount THEN
	RemoteDevice();
END_IF
(* remind current number of update counter *)
_nUpdateCount := RemoteDevice._nUpdateCount;

IF RemoteDevice.bFirstCycle THEN
	(* first call of the server device since reboot/reset *)
	bReady := FALSE;

ELSIF NOT RemoteDevice.bOperational THEN
	nErrorId := BACnet_ERR_OPERATIONAL;
	bReady := FALSE;

ELSIF _StatusFlags >= 4 THEN
	(* clear error flag *)
	nErrorId := BACnet_ERR_NO_ERROR;
	(* ready state *)
	bReady := TRUE;

	(* present value *)
	bPresentValue := F_BinPV_To_Bool(_PresentValue);

	(* build bit states *)
	_StatusFlagsBits := F_BACnet_StatusFlags(_StatusFlags);

	(* copy states to output *)
	bOverridden := _StatusFlagsBits.overridden;
	bOutOfService := _StatusFlagsBits.out_of_service;
	bFault := _StatusFlagsBits.fault;
	bInAlarm := _StatusFlagsBits.in_alarm;

ELSE
	(* server device not ready, reset local ready also *)
	bReady := FALSE;
	(* and set error ID *)
	nErrorId := BACnet_ERR_WRONG_MAPPING;
END_IF

(* set error flag *)
bError := (nErrorId <> BACnet_ERR_NO_ERROR);
END_FUNCTION_BLOCK

(* POU FB_BACnet_RemoteBinaryValue_EX, ST *)
FUNCTION_BLOCK FB_BACnet_RemoteBinaryValue_EX
VAR_INPUT
	bEnablePV			: BOOL; (* enable present value with priority x in priority array, FALSE = priority x disable *)
	bNullPV				: BOOL; (* clear priority entry *)
	bPV					: BOOL; (* present value bool type *)
END_VAR
VAR_IN_OUT
	RemoteDevice		: FB_BACnet_RemoteDevice;
END_VAR
VAR_OUTPUT
	bReady				: BOOL;
	bPresentValue		: BOOL;
	bOverridden			: BOOL;
	bOutOfService		: BOOL;
	bFault				: BOOL;
	bInAlarm			: BOOL;
	bOtherFault			: BOOL;
	eEventState			: E_BACNETEVENTSTATE;
	nChangeOfState		: UDINT;
	tObjectID			: T_BACnet_ObjectIdentifier := 16#FFFFFFFF;
	bError				: BOOL;
	nErrorId			: UINT;
END_VAR
VAR
	_ChangeOfStateCount AT%I*: UDINT;	(* ~(BACnet_ChangeOfStateCount			:		: ) *)
	_ObjectId AT%I*: DWORD;				(* ~(BACnet_ObjectIdentifier			:		: LINK) *)
	_PresentValue AT%I*: WORD; 			(* ~(BACnet_PresentValue 				:		: )
								   			(BACnet_ObjectType 					: BV	: )
											(BACnet_RemoteCycletimeRead 		: 1000	: )
											(BACnet_RemoteFlagsRead        		: 1		: )
											(BACnet_RemoteResubscriptionInterval: 240	: )
	                                		(BACnet_RemoteCycleTimeWrite   		: 1000	: )
	                                		(BACnet_RemoteFlagsWrite       		: 1		: )	*)
	_StatusFlags AT%I*: WORD; 			(* ~(BACnet_StatusFlags 				:		: )	*)
	_Reliability AT%I*: WORD;			(* ~(BACnet_Reliability 				:		: )	*)
	_EventState AT%I*: WORD;			(* ~(BACnet_EventState					:		: )	*)
    _PresentValue_Priority12 AT%Q*: WORD;(* ~(BACnet_PresentValue_Priority12	:		: )	*)
	_nUpdateCount : UDINT := 0;
	_StatusFlagsBits : ST_BACnet_StatusFlags;
END_VAR
(* update client device *)
IF RemoteDevice._nUpdateCount = _nUpdateCount THEN
	RemoteDevice();
END_IF
(* remind current number of update counter *)
_nUpdateCount := RemoteDevice._nUpdateCount;

IF RemoteDevice.bFirstCycle THEN
	(* first call of the server device since reboot/reset *)
	bReady := FALSE;
	_PresentValue_Priority12 := BACnetBinaryPV_Nothing;
ELSIF NOT RemoteDevice.bOperational THEN
	nErrorId := BACnet_ERR_OPERATIONAL;
	bReady := FALSE;

ELSIF (F_BACnet_GetObjType(_ObjectId) <> BACnetObjectType_BinaryValue) THEN
	(* wrong mapping / invalid object ID *)
	IF _ObjectId = 0 THEN
		nErrorId := BACnet_ERR_WRONG_MAPPING;
	ELSE
		nErrorId := BACnet_ERR_INVALID_OBJECTID;
	END_IF
	bReady := FALSE;
	tObjectID := 16#FFFFFFFF;

ELSIF _StatusFlags >= 4 THEN
	(* clear error flag *)
	nErrorId := BACnet_ERR_NO_ERROR;
	(* ready state *)
	bReady := TRUE;

	(* write into priority array *)
	_PresentValue_Priority12 := F_Bool_To_BinPV(bEnablePV, bNullPV, bPV);

	(* present value *)
	bPresentValue := F_BinPV_To_Bool(_PresentValue);

	(* build bit states *)
	_StatusFlagsBits := F_BACnet_StatusFlags(_StatusFlags);

	(* copy states to output *)
	bOverridden := _StatusFlagsBits.overridden;
	bOutOfService := _StatusFlagsBits.out_of_service;
	bFault := _StatusFlagsBits.fault;
	bInAlarm := _StatusFlagsBits.in_alarm;
	bOtherFault := (_Reliability = BACnetReliability_unreliable_other);
	eEventState := _EventState;
	tObjectID := _ObjectId;

	(* copy change_of_state_count *)
	nChangeOfState := _ChangeOfStateCount;

ELSE
	(* server device not ready, reset local ready also *)
	bReady := FALSE;
	(* and set error ID *)
	nErrorId := BACnet_ERR_WRONG_MAPPING;
END_IF

(* set error flag *)
bError := (nErrorId <> BACnet_ERR_NO_ERROR);
END_FUNCTION_BLOCK

(* POU FB_BACnet_RemoteBinaryValue_WR, ST *)
FUNCTION_BLOCK FB_BACnet_RemoteBinaryValue_WR
VAR_INPUT
	bEnablePV			: BOOL; (* enable present value with priority x in priority array, FALSE = priority x disable *)
	bNullPV				: BOOL; (* clear priority entry *)
	bPV					: BOOL; (* present value bool type *)
END_VAR
VAR_IN_OUT
	RemoteDevice		: FB_BACnet_RemoteDevice;
END_VAR
VAR_OUTPUT
	bReady				: BOOL;
	bPresentValue		: BOOL;
	bOverridden			: BOOL;
	bOutOfService		: BOOL;
	bFault				: BOOL;
	bInAlarm			: BOOL;
	bError				: BOOL;
	nErrorId			: UINT;
END_VAR
VAR

	_PresentValue AT%I*: WORD; 			(* ~(BACnet_PresentValue 				:		: )
								   			(BACnet_ObjectType 					: BV	: )
											(BACnet_RemoteCycletimeRead 		: 1000	: )
											(BACnet_RemoteFlagsRead        		: 1		: )
											(BACnet_RemoteResubscriptionInterval: 240	: )
	                                		(BACnet_RemoteCycleTimeWrite   		: 1000	: )
	                                		(BACnet_RemoteFlagsWrite       		: 1		: )	*)
    _PresentValue_Priority12 AT%Q*: WORD;(* ~(BACnet_PresentValue_Priority12	:		: )	*)
	_StatusFlags AT%I*: WORD; 			(* ~(BACnet_StatusFlags 				:		: )	*)
	_StatusFlagsBits : ST_BACnet_StatusFlags;

	_nUpdateCount : UDINT := 0;
END_VAR
(* update client device *)
IF RemoteDevice._nUpdateCount = _nUpdateCount THEN
	RemoteDevice();
END_IF
(* remind current number of update counter *)
_nUpdateCount := RemoteDevice._nUpdateCount;

IF RemoteDevice.bFirstCycle THEN
	(* first call of the server device since reboot/reset *)
	bReady := FALSE;
	_PresentValue_Priority12 := BACnetBinaryPV_Nothing;
ELSIF NOT RemoteDevice.bOperational THEN
	nErrorId := BACnet_ERR_OPERATIONAL;
	bReady := FALSE;

ELSIF _StatusFlags >= 4 THEN
	(* clear error flag *)
	nErrorId := BACnet_ERR_NO_ERROR;
	(* ready state *)
	bReady := TRUE;

	(* write into priority array *)
	_PresentValue_Priority12 := F_Bool_To_BinPV(bEnablePV, bNullPV, bPV);

	(* present value *)
	bPresentValue := F_BinPV_To_Bool(_PresentValue);

	(* build bit states *)
	_StatusFlagsBits := F_BACnet_StatusFlags(_StatusFlags);

	(* copy states to output *)
	bOverridden := _StatusFlagsBits.overridden;
	bOutOfService := _StatusFlagsBits.out_of_service;
	bFault := _StatusFlagsBits.fault;
	bInAlarm := _StatusFlagsBits.in_alarm;

ELSE
	(* server device not ready, reset local ready also *)
	bReady := FALSE;
	(* and set error ID *)
	nErrorId := BACnet_ERR_WRONG_MAPPING;
END_IF

(* set error flag *)
bError := (nErrorId <> BACnet_ERR_NO_ERROR);
END_FUNCTION_BLOCK

(* POU FB_BACnet_RemoteCalendar, ST *)
FUNCTION_BLOCK FB_BACnet_RemoteCalendar
VAR_IN_OUT
	RemoteDevice		: FB_BACnet_RemoteDevice;
END_VAR
VAR_OUTPUT
	bReady				: BOOL;
	bPresentValue		: BOOL;
	bError				: BOOL;
	nErrorId			: UINT;
END_VAR
VAR
	_PresentValue AT%I*: BOOL;	(* ~(BACnet_PresentValue 				:		: )
									(BACnet_ObjectType 					: CAL	: )
									(BACnet_RemoteCycletimeRead 		: 1000	: )
									(BACnet_RemoteFlagsRead        		: 1		: )
									(BACnet_RemoteResubscriptionInterval: 240	: )
                            		(BACnet_RemoteCycleTimeWrite   		: 1000	: )
                            		(BACnet_RemoteFlagsWrite       		: 1		: )	*)
	_nUpdateCount : UDINT := 0;
END_VAR
(* update client device *)
IF RemoteDevice._nUpdateCount = _nUpdateCount THEN
	RemoteDevice();
END_IF
(* remind current number of update counter *)
_nUpdateCount := RemoteDevice._nUpdateCount;

IF RemoteDevice.bOperational THEN
	(* clear error flag *)
	nErrorId := BACnet_ERR_NO_ERROR;
	(* ready state *)
	bReady := TRUE;
	(* present value *)
	bPresentValue := _PresentValue;
ELSE
	(* server device not ready, reset local ready also *)
	bReady := FALSE;
	(* and set error ID *)
	nErrorId := BACnet_ERR_OPERATIONAL;
END_IF

(* set error flag *)
bError := (nErrorId <> BACnet_ERR_NO_ERROR);
END_FUNCTION_BLOCK

(* POU FB_BACnet_RemoteCalendar_EX, ST *)
FUNCTION_BLOCK FB_BACnet_RemoteCalendar_EX
VAR_IN_OUT
	RemoteDevice		: FB_BACnet_RemoteDevice;
END_VAR
VAR_OUTPUT
	bReady				: BOOL;
	bPresentValue		: BOOL;
	tObjectID			: T_BACnet_ObjectIdentifier := 16#FFFFFFFF;
	bError				: BOOL;
	nErrorId			: UINT;
END_VAR
VAR
	_PresentValue AT%I*: BOOL;	(* ~(BACnet_PresentValue 				:		: )
									(BACnet_ObjectType 					: CAL	: )
									(BACnet_RemoteCycletimeRead 		: 1000	: )
									(BACnet_RemoteFlagsRead        		: 1		: )
									(BACnet_RemoteResubscriptionInterval: 240	: )
                            		(BACnet_RemoteCycleTimeWrite   		: 1000	: )
                            		(BACnet_RemoteFlagsWrite       		: 1		: )	*)
	_ObjectId AT%I*: DWORD;		(* ~(BACnet_ObjectIdentifier			:		: LINK) *)
	_nUpdateCount : UDINT := 0;
END_VAR
(* update client device *)
IF RemoteDevice._nUpdateCount = _nUpdateCount THEN
	RemoteDevice();
END_IF
(* remind current number of update counter *)
_nUpdateCount := RemoteDevice._nUpdateCount;

IF NOT RemoteDevice.bOperational THEN
	nErrorId := BACnet_ERR_OPERATIONAL;
	bReady := FALSE;

ELSIF (F_BACnet_GetObjType(_ObjectId) <> BACnetObjectType_Calendar) THEN
	(* wrong mapping / invalid object ID *)
	IF _ObjectId = 0 THEN
		nErrorId := BACnet_ERR_WRONG_MAPPING;
	ELSE
		nErrorId := BACnet_ERR_INVALID_OBJECTID;
	END_IF
	bReady := FALSE;
	tObjectID := 16#FFFFFFFF;

ELSE
	(* clear error flag *)
	nErrorId := BACnet_ERR_NO_ERROR;
	(* ready state *)
	bReady := TRUE;
	(* present value *)
	bPresentValue := _PresentValue;
	tObjectID := _ObjectId;

END_IF

(* set error flag *)
bError := (nErrorId <> BACnet_ERR_NO_ERROR);
END_FUNCTION_BLOCK

(* POU FB_BACnet_RemoteCommand, ST *)
FUNCTION_BLOCK FB_BACnet_RemoteCommand
VAR_IN_OUT
	RemoteDevice		: FB_BACnet_RemoteDevice;
END_VAR
VAR_OUTPUT
	bReady				: BOOL;
	nPresentValue		: UDINT;
	bAllWritesOk		: BOOL; (* all actions in selected action list are written *)
	bInProcess			: BOOL; (* object is busy *)
	bError				: BOOL;
	nErrorId			: UINT;
END_VAR
VAR
	_PresentValueIn AT%I*: UDINT; 		(* ~(BACnet_PresentValue 				:		: )
								   			(BACnet_ObjectType 					: CMD	: )
											(BACnet_RemoteCycletimeRead 		: 1000	: )
											(BACnet_RemoteFlagsRead        		: 1		: )
											(BACnet_RemoteResubscriptionInterval: 240	: )
	                                		(BACnet_RemoteCycleTimeWrite   		: 1000	: )
	                                		(BACnet_RemoteFlagsWrite       		: 1		: )	*)
	_InProcess AT%I*: BOOL;				(* ~(BACnet_InProcess 					:		: )	*)
	_AllWritesSuccessful AT%I*: BOOL;	(* ~(BACnet_AllWritesSuccessful			:		: )	*)
	_nUpdateCount : UDINT := 0;
	_rtrigRetriggerPv : R_TRIG;
END_VAR
(* update client device *)
IF RemoteDevice._nUpdateCount = _nUpdateCount THEN
	RemoteDevice();
END_IF
(* remind current number of update counter *)
_nUpdateCount := RemoteDevice._nUpdateCount;

IF RemoteDevice.bOperational THEN
	(* clear error flag *)
	nErrorId := BACnet_ERR_NO_ERROR;
	(* ready state *)
	bReady := TRUE;
	(* present value from BACnet *)
	nPresentValue := _PresentValueIn;

	(* other states *)
	bAllWritesOk := _AllWritesSuccessful;
	bInProcess := _InProcess;
ELSIF RemoteDevice.bFirstCycle THEN
	(* first call of the server device since reboot/reset *)
	bReady := FALSE;
ELSE
	(* server device not ready, reset local ready also *)
	bReady := FALSE;
	(* and set error ID *)
	nErrorId := BACnet_ERR_WRONG_MAPPING;
END_IF

(* set error flag *)
bError := (nErrorId <> BACnet_ERR_NO_ERROR);
END_FUNCTION_BLOCK

(* POU FB_BACnet_RemoteCommand_EX, ST *)
FUNCTION_BLOCK FB_BACnet_RemoteCommand_EX
VAR_INPUT
	bEnablePV			: BOOL;
	nPV					: UDINT;
	bRetrigger			: BOOL; (* execute selected action on raising edge again *)
END_VAR
VAR_IN_OUT
	RemoteDevice		: FB_BACnet_RemoteDevice;
END_VAR
VAR_OUTPUT
	bReady				: BOOL;
	nPresentValue		: UDINT;
	bAllWritesOk		: BOOL; (* all actions in selected action list are written *)
	bInProcess			: BOOL; (* object is busy *)
	tObjectID			: T_BACnet_ObjectIdentifier := 16#FFFFFFFF;
	bError				: BOOL;
	nErrorId			: UINT;
END_VAR
VAR
	_PresentValueIn AT%I*: UDINT; 		(* ~(BACnet_PresentValue 				:		: )
								   			(BACnet_ObjectType 					: CMD	: )
											(BACnet_RemoteCycletimeRead 		: 1000	: )
											(BACnet_RemoteFlagsRead        		: 1		: )
											(BACnet_RemoteResubscriptionInterval: 240	: )
	                                		(BACnet_RemoteCycleTimeWrite   		: 1000	: )
	                                		(BACnet_RemoteFlagsWrite       		: 1		: )	*)
	_ObjectId AT%I*: DWORD;				(* ~(BACnet_ObjectIdentifier			:		: LINK) *)
	_InProcess AT%I*: BOOL;				(* ~(BACnet_InProcess 					:		: )	*)
	_AllWritesSuccessful AT%I*: BOOL;	(* ~(BACnet_AllWritesSuccessful			:		: )	*)
    _PresentValueOut AT%Q*: UDINT;		(* ~(BACnet_PresentValue	 	   		:      	: )	*)
	_nUpdateCount : UDINT := 0;
	_rtrigRetriggerPv : R_TRIG;
	_bRetriggerReq : BOOL;
END_VAR
(* update client device *)
IF RemoteDevice._nUpdateCount = _nUpdateCount THEN
	RemoteDevice();
END_IF
(* remind current number of update counter *)
_nUpdateCount := RemoteDevice._nUpdateCount;

(* call trigger *)
_rtrigRetriggerPv(CLK:= bRetrigger, Q=> );

IF RemoteDevice.bFirstCycle THEN
	(* first call of the server device since reboot/reset *)
	bReady := FALSE;
	_PresentValueOut := 0;
	_bRetriggerReq := FALSE;

ELSIF NOT RemoteDevice.bOperational THEN
	(* server device not ready, reset local ready also *)
	bReady := FALSE;
	(* and set error ID *)
	nErrorId := BACnet_ERR_WRONG_MAPPING;
	_bRetriggerReq := FALSE;

ELSIF (F_BACnet_GetObjType(_ObjectId) <> BACnetObjectType_Command) THEN
	(* wrong mapping / invalid object ID *)
	IF _ObjectId = 0 THEN
		nErrorId := BACnet_ERR_WRONG_MAPPING;
	ELSE
		nErrorId := BACnet_ERR_INVALID_OBJECTID;
	END_IF
	bReady := FALSE;
	tObjectID := 16#FFFFFFFF;
	_bRetriggerReq := FALSE;

ELSE
	(* object ID *)
	tObjectID := _ObjectId;
	(* clear error flag *)
	nErrorId := BACnet_ERR_NO_ERROR;
	(* activities *)
	bAllWritesOk := _AllWritesSuccessful;
	bInProcess := _InProcess;
	(* ready state *)
	bReady := TRUE;
	(* present value from BACnet *)
	nPresentValue := _PresentValueIn;
	(* present value to BACnet *)
	IF bEnablePV THEN
		IF (NOT bInProcess) THEN
			IF _bRetriggerReq THEN
				(* trigger action list *)
				_PresentValueOut := 0;
			ELSE
				(* set present value *)
				_PresentValueOut := nPV;
			END_IF
			_bRetriggerReq := FALSE;
		END_IF
	ELSE
		(* deactivate mapped present value --> other objects can write to property *)
		_PresentValueOut := 16#0;
		_bRetriggerReq := FALSE;
	END_IF

END_IF

(* set error flag *)
bError := (nErrorId <> BACnet_ERR_NO_ERROR);
END_FUNCTION_BLOCK

(* POU FB_BACnet_RemoteCommand_WR, ST *)
FUNCTION_BLOCK FB_BACnet_RemoteCommand_WR
VAR_INPUT
	bEnablePV			: BOOL;
	nPV					: UDINT;
	bRetrigger			: BOOL; (* execute selected action on raising edge again *)
END_VAR
VAR_IN_OUT
	RemoteDevice		: FB_BACnet_RemoteDevice;
END_VAR
VAR_OUTPUT
	bReady				: BOOL;
	nPresentValue		: UDINT;
	bAllWritesOk		: BOOL; (* all actions in selected action list are written *)
	bInProcess			: BOOL; (* object is busy *)
	bError				: BOOL;
	nErrorId			: UINT;
END_VAR
VAR
	_PresentValueIn AT%I*: UDINT; 		(* ~(BACnet_PresentValue 				:		: )
								   			(BACnet_ObjectType 					: CMD	: )
											(BACnet_RemoteCycletimeRead 		: 1000	: )
											(BACnet_RemoteFlagsRead        		: 1		: )
											(BACnet_RemoteResubscriptionInterval: 240	: )
	                                		(BACnet_RemoteCycleTimeWrite   		: 1000	: )
	                                		(BACnet_RemoteFlagsWrite       		: 1		: )	*)
	_InProcess AT%I*: BOOL;				(* ~(BACnet_InProcess 					:		: )	*)
	_AllWritesSuccessful AT%I*: BOOL;	(* ~(BACnet_AllWritesSuccessful			:		: )	*)
    _PresentValueOut AT%Q*: UDINT;		(* ~(BACnet_PresentValue	 	   		:      	: )	*)
	_nUpdateCount : UDINT := 0;
	_rtrigRetriggerPv : R_TRIG;
END_VAR
(* update client device *)
IF RemoteDevice._nUpdateCount = _nUpdateCount THEN
	RemoteDevice();
END_IF
(* remind current number of update counter *)
_nUpdateCount := RemoteDevice._nUpdateCount;

(* call trigger *)
_rtrigRetriggerPv(CLK:= bRetrigger, Q=> );

IF RemoteDevice.bOperational THEN
	(* clear error flag *)
	nErrorId := BACnet_ERR_NO_ERROR;
	(* ready state *)
	bReady := TRUE;
	(* present value from BACnet *)
	nPresentValue := _PresentValueIn;
	(* present value to BACnet *)
	IF bEnablePV THEN
		IF _rtrigRetriggerPv.Q THEN
			(* trigger action list *)
			_PresentValueOut := 0;
		ELSE
			(* set present value *)
			_PresentValueOut := nPV;
		END_IF
	ELSE
		(* deactivate mapped present value --> other objects can write to property *)
		_PresentValueOut := 16#0;
	END_IF
	(* other states *)
	bAllWritesOk := _AllWritesSuccessful;
	bInProcess := _InProcess;
ELSIF RemoteDevice.bFirstCycle THEN
	(* first call of the server device since reboot/reset *)
	bReady := FALSE;
	_PresentValueOut := 0;
ELSE
	(* server device not ready, reset local ready also *)
	bReady := FALSE;
	(* and set error ID *)
	nErrorId := BACnet_ERR_WRONG_MAPPING;
END_IF

(* set error flag *)
bError := (nErrorId <> BACnet_ERR_NO_ERROR);
END_FUNCTION_BLOCK

(* POU FB_BACnet_RemoteEventEnrollment, ST *)
FUNCTION_BLOCK FB_BACnet_RemoteEventEnrollment
VAR_IN_OUT
	RemoteDevice		: FB_BACnet_RemoteDevice;
END_VAR
VAR_OUTPUT
	bReady				: BOOL;
	bError				: BOOL;
	nErrorId			: UINT;
END_VAR
VAR
	_ObjectType: E_BACNETOBJECTTYPE;	(* ~ (BACNET_OBJECTTYPE : EE : )	*)
	_nUpdateCount : UDINT := 0;
END_VAR
_ObjectType := BACnetObjectType_EventEnrollment;
(* update client device *)
IF RemoteDevice._nUpdateCount = _nUpdateCount THEN
	RemoteDevice();
END_IF
(* remind current number of update counter *)
_nUpdateCount := RemoteDevice._nUpdateCount;

IF RemoteDevice.bOperational THEN
	(* clear error flag *)
	nErrorId := BACnet_ERR_NO_ERROR;
	(* ready state *)
	bReady := TRUE;
ELSE
	(* server device not ready, reset local ready also *)
	bReady := FALSE;
	(* and set error ID *)
	nErrorId := BACnet_ERR_OPERATIONAL;
END_IF

(* set error flag *)
bError := (nErrorId <> BACnet_ERR_NO_ERROR);
END_FUNCTION_BLOCK

(* POU FB_BACnet_RemoteEventEnrollment_EX, ST *)
FUNCTION_BLOCK FB_BACnet_RemoteEventEnrollment_EX
VAR_IN_OUT
	RemoteDevice		: FB_BACnet_RemoteDevice;
END_VAR
VAR_OUTPUT
	bReady				: BOOL;
	tObjectID			: T_BACnet_ObjectIdentifier := 16#FFFFFFFF;
	bError				: BOOL;
	nErrorId			: UINT;
END_VAR
VAR
	_ObjectId AT%I*: DWORD;	(* ~(BACnet_ObjectIdentifier:		: LINK)
								(BACNET_OBJECTTYPE		: EE	: ) *)
	_nUpdateCount : UDINT := 0;
END_VAR
(* update client device *)
IF RemoteDevice._nUpdateCount = _nUpdateCount THEN
	RemoteDevice();
END_IF
(* remind current number of update counter *)
_nUpdateCount := RemoteDevice._nUpdateCount;

IF NOT RemoteDevice.bOperational THEN
	(* server device not ready, reset local ready also *)
	bReady := FALSE;
	(* and set error ID *)
	nErrorId := BACnet_ERR_OPERATIONAL;

ELSIF (F_BACnet_GetObjType(_ObjectId) <> BACnetObjectType_EventEnrollment) THEN
	(* wrong mapping / invalid object ID *)
	IF _ObjectId = 0 THEN
		nErrorId := BACnet_ERR_WRONG_MAPPING;
	ELSE
		nErrorId := BACnet_ERR_INVALID_OBJECTID;
	END_IF
	bReady := FALSE;
	tObjectID := 16#FFFFFFFF;

ELSE
	(* clear error flag *)
	nErrorId := BACnet_ERR_NO_ERROR;
	(* ready state *)
	bReady := TRUE;
	tObjectID := _ObjectId;

END_IF

(* set error flag *)
bError := (nErrorId <> BACnet_ERR_NO_ERROR);
END_FUNCTION_BLOCK

(* POU FB_BACnet_RemoteEventLog, ST *)
FUNCTION_BLOCK FB_BACnet_RemoteEventLog
VAR_IN_OUT
	RemoteDevice			: FB_BACnet_RemoteDevice;
END_VAR
VAR_OUTPUT
	bReady				: BOOL;
	bLogEnable			: BOOL;
	nRecordCount		: UDINT;
	nTotalCount			: UDINT;
	bError				: BOOL;
	nErrorId			: UINT;
END_VAR
VAR
	_RecordCount AT%I*: UDINT;		(* ~(BACnet_RecordCount					:		: )
										(BACnet_ObjectType					: ELOG	: )
										(BACnet_RemoteCycletimeRead 		: 1000	: )
										(BACnet_RemoteFlagsRead        		: 1		: )
										(BACnet_RemoteResubscriptionInterval: 240	: )
                                		(BACnet_RemoteCycleTimeWrite   		: 1000	: )
                                		(BACnet_RemoteFlagsWrite       		: 1		: )	*)
	_TotalRecordCount AT%I*: UDINT;	(* ~(BACnet_TotalRecordCount			:		: )	*)
	_LogEnable AT%I*: BOOL;			(* ~(BACnet_LogEnable					: 		: )	*)
	_nUpdateCount : UDINT := 0;
END_VAR
(* update client device *)
IF RemoteDevice._nUpdateCount = _nUpdateCount THEN
	RemoteDevice();
END_IF
(* remind current number of update counter *)
_nUpdateCount := RemoteDevice._nUpdateCount;

IF RemoteDevice.bOperational THEN
	(* clear error flag *)
	nErrorId := BACnet_ERR_NO_ERROR;
	(* ready state *)
	bReady := TRUE;

	(* other states *)
	nRecordCount := _RecordCount;
	nTotalCount := _TotalRecordCount;
	bLogEnable := _LogEnable;

ELSE
	bReady := FALSE;
	(* and set error ID *)
	nErrorId := BACnet_ERR_OPERATIONAL;
END_IF

(* set error flag *)
bError := (nErrorId <> BACnet_ERR_NO_ERROR);
END_FUNCTION_BLOCK

(* POU FB_BACnet_RemoteEventLog_EX, ST *)
FUNCTION_BLOCK FB_BACnet_RemoteEventLog_EX
VAR_OUTPUT
	bReady				: BOOL;
	bLogEnable			: BOOL;
	nRecordCount		: UDINT;
	nTotalCount			: UDINT;
	eEventState			: E_BACNETEVENTSTATE;
	tObjectID			: T_BACnet_ObjectIdentifier := 16#FFFFFFFF;
	bError				: BOOL;
	nErrorId			: UINT;
END_VAR
VAR_IN_OUT
	RemoteDevice			: FB_BACnet_RemoteDevice;
END_VAR
VAR
	_RecordCount AT%I*: UDINT;			(* ~(BACnet_RecordCount					:		: )
											(BACnet_ObjectType					: ELOG	: )
											(BACnet_RemoteCycletimeRead 		: 1000	: )
											(BACnet_RemoteFlagsRead        		: 1		: )
											(BACnet_RemoteResubscriptionInterval: 240	: )
											(BACnet_RemoteCycleTimeWrite   		: 1000	: )
                                			(BACnet_RemoteFlagsWrite       		: 1		: )	*)
	_TotalRecordCount AT%I*: UDINT;		(* ~(BACnet_TotalRecordCount			:		: )	*)
	_ObjectId AT%I*: DWORD;				(* ~(BACnet_ObjectIdentifier			:		: LINK) *)
	_EventState AT%I*: WORD;			(* ~(BACnet_EventState					:		: )	*)
	_LogEnable AT%I*: BOOL;				(* ~(BACnet_LogEnable					: 		: )	*)
	_nUpdateCount : UDINT := 0;
END_VAR
(* update client device *)
IF RemoteDevice._nUpdateCount = _nUpdateCount THEN
	RemoteDevice();
END_IF
(* remind current number of update counter *)
_nUpdateCount := RemoteDevice._nUpdateCount;

IF NOT RemoteDevice.bOperational THEN
	(* mapping seems to be wrong *)
	nErrorId := BACnet_ERR_OPERATIONAL;
	bReady := FALSE;

ELSIF (F_BACnet_GetObjType(_ObjectId) <> BACnetObjectType_EventLog) THEN
	(* wrong mapping / invalid object ID *)
	IF _ObjectId = 0 THEN
		nErrorId := BACnet_ERR_WRONG_MAPPING;
	ELSE
		nErrorId := BACnet_ERR_INVALID_OBJECTID;
	END_IF
	bReady := FALSE;
	tObjectID := 16#FFFFFFFF;

ELSIF _EventState >= 0 THEN
	(* clear error flag *)
	nErrorId := BACnet_ERR_NO_ERROR;
	(* ready state *)
	bReady := TRUE;

	(* convert enumeration *)
	eEventState := _EventState;

	(* other states *)
	nRecordCount := _RecordCount;
	nTotalCount := _TotalRecordCount;
	bLogEnable := _LogEnable;
	tObjectID := _ObjectId;

ELSE
	bReady := FALSE;
	(* and set error ID *)
	nErrorId := BACnet_ERR_WRONG_MAPPING;
END_IF

(* set error flag *)
bError := (nErrorId <> BACnet_ERR_NO_ERROR);
END_FUNCTION_BLOCK

(* POU FB_BACnet_RemoteFile, ST *)
FUNCTION_BLOCK FB_BACnet_RemoteFile
VAR_IN_OUT
	RemoteDevice		: FB_BACnet_RemoteDevice;
END_VAR
VAR_OUTPUT
	bReady				: BOOL;
	fFileSize			: UDINT;
	bError				: BOOL;
	nErrorId			: UINT;
END_VAR
VAR
	_FileSize 			AT%I*: UDINT; 	(* ~(BACnet_FileSize 					:		: )
					   						(BACnet_ObjectType 					: FILE	: )
											(BACnet_RemoteCycletimeRead 		: 1000	: )
											(BACnet_RemoteFlagsRead        		: 1		: )
											(BACnet_RemoteResubscriptionInterval: 240	: )
	                                		(BACnet_RemoteCycleTimeWrite   		: 1000	: )
	                                		(BACnet_RemoteFlagsWrite       		: 1		: )	*)
	_nUpdateCount		: UDINT := 0;
END_VAR
(* update client device *)
IF RemoteDevice._nUpdateCount = _nUpdateCount THEN
	RemoteDevice();
END_IF
(* remind current number of update counter *)
_nUpdateCount := RemoteDevice._nUpdateCount;

IF RemoteDevice.bOperational THEN
	(* clear error flag *)
	nErrorId := BACnet_ERR_NO_ERROR;
	(* ready state *)
	bReady := TRUE;
	fFileSize := _FileSize;
ELSE
	(* server device not ready, reset local ready also *)
	bReady := FALSE;
	(* and set error ID *)
	nErrorId := BACnet_ERR_OPERATIONAL;
END_IF

(* set error flag *)
bError := (nErrorId <> BACnet_ERR_NO_ERROR);
END_FUNCTION_BLOCK

(* POU FB_BACnet_RemoteFile_EX, ST *)
FUNCTION_BLOCK FB_BACnet_RemoteFile_EX
VAR_IN_OUT
	RemoteDevice		: FB_BACnet_RemoteDevice;
END_VAR
VAR_OUTPUT
	bReady				: BOOL;
	fFileSize			: UDINT;
	tObjectID			: T_BACnet_ObjectIdentifier := 16#FFFFFFFF;
	bError				: BOOL;
	nErrorId			: UINT;
END_VAR
VAR
	_FileSize 			AT%I*: UDINT; 	(* ~(BACnet_FileSize 					:		: )
					   						(BACnet_ObjectType 					: FILE	: )
											(BACnet_RemoteCycletimeRead 		: 1000	: )
											(BACnet_RemoteFlagsRead        		: 1		: )
											(BACnet_RemoteResubscriptionInterval: 240	: )
	                                		(BACnet_RemoteCycleTimeWrite   		: 1000	: )
	                                		(BACnet_RemoteFlagsWrite       		: 1		: )	*)
	_ObjectId AT%I*: DWORD;				(* ~(BACnet_ObjectIdentifier			:		: LINK) *)
	_nUpdateCount		: UDINT := 0;
END_VAR
(* update client device *)
IF RemoteDevice._nUpdateCount = _nUpdateCount THEN
	RemoteDevice();
END_IF
(* remind current number of update counter *)
_nUpdateCount := RemoteDevice._nUpdateCount;

IF NOT RemoteDevice.bOperational THEN
	(* server device not ready, reset local ready also *)
	bReady := FALSE;
	(* and set error ID *)
	nErrorId := BACnet_ERR_OPERATIONAL;

ELSIF (F_BACnet_GetObjType(_ObjectId) <> BACnetObjectType_File) THEN
	(* wrong mapping / invalid object ID *)
	IF _ObjectId = 0 THEN
		nErrorId := BACnet_ERR_WRONG_MAPPING;
	ELSE
		nErrorId := BACnet_ERR_INVALID_OBJECTID;
	END_IF
	bReady := FALSE;
	tObjectID := 16#FFFFFFFF;

ELSE
	(* clear error flag *)
	nErrorId := BACnet_ERR_NO_ERROR;
	(* ready state *)
	bReady := TRUE;
	fFileSize := _FileSize;
	tObjectID := _ObjectId;

END_IF

(* set error flag *)
bError := (nErrorId <> BACnet_ERR_NO_ERROR);
END_FUNCTION_BLOCK

(* POU FB_BACnet_RemoteGroup, ST *)
FUNCTION_BLOCK FB_BACnet_RemoteGroup
VAR_IN_OUT
	RemoteDevice		: FB_BACnet_RemoteDevice;
END_VAR
VAR_OUTPUT
	bReady				: BOOL;
	bError				: BOOL;
	nErrorId			: UINT;
END_VAR
VAR
	_ObjectType: E_BACNETOBJECTTYPE;	(* ~ (BACNET_OBJECTTYPE : GROUP : )	*)
	_nUpdateCount : UDINT := 0;
END_VAR
_ObjectType := BACnetObjectType_Group;
(* update client device *)
IF RemoteDevice._nUpdateCount = _nUpdateCount THEN
	RemoteDevice();
END_IF
(* remind current number of update counter *)
_nUpdateCount := RemoteDevice._nUpdateCount;

IF RemoteDevice.bOperational THEN
	(* clear error flag *)
	nErrorId := BACnet_ERR_NO_ERROR;
	(* ready state *)
	bReady := TRUE;
ELSE
	(* server device not ready, reset local ready also *)
	bReady := FALSE;
	(* and set error ID *)
	nErrorId := BACnet_ERR_OPERATIONAL;
END_IF

(* set error flag *)
bError := (nErrorId <> BACnet_ERR_NO_ERROR);
END_FUNCTION_BLOCK

(* POU FB_BACnet_RemoteGroup_EX, ST *)
FUNCTION_BLOCK FB_BACnet_RemoteGroup_EX
VAR_IN_OUT
	RemoteDevice		: FB_BACnet_RemoteDevice;
END_VAR
VAR_OUTPUT
	bReady				: BOOL;
	tObjectID			: T_BACnet_ObjectIdentifier := 16#FFFFFFFF;
	bError				: BOOL;
	nErrorId			: UINT;
END_VAR
VAR
	_ObjectId AT%I*: DWORD;			(* ~(BACnet_ObjectIdentifier:		: LINK)
										(BACNET_OBJECTTYPE		: GROUP : ) *)
	_nUpdateCount : UDINT := 0;
END_VAR
(* update client device *)
IF RemoteDevice._nUpdateCount = _nUpdateCount THEN
	RemoteDevice();
END_IF
(* remind current number of update counter *)
_nUpdateCount := RemoteDevice._nUpdateCount;

IF NOT RemoteDevice.bOperational THEN
	(* server device not ready, reset local ready also *)
	bReady := FALSE;
	(* and set error ID *)
	nErrorId := BACnet_ERR_OPERATIONAL;

ELSIF (F_BACnet_GetObjType(_ObjectId) <> BACnetObjectType_Group) THEN
	(* wrong mapping / invalid object ID *)
	IF _ObjectId = 0 THEN
		nErrorId := BACnet_ERR_WRONG_MAPPING;
	ELSE
		nErrorId := BACnet_ERR_INVALID_OBJECTID;
	END_IF
	bReady := FALSE;
	tObjectID := 16#FFFFFFFF;

ELSE
	(* clear error flag *)
	nErrorId := BACnet_ERR_NO_ERROR;
	(* ready state *)
	bReady := TRUE;
	tObjectID := _ObjectId;
END_IF

(* set error flag *)
bError := (nErrorId <> BACnet_ERR_NO_ERROR);
END_FUNCTION_BLOCK

(* POU FB_BACnet_RemoteLoop, ST *)
FUNCTION_BLOCK FB_BACnet_RemoteLoop
VAR_IN_OUT
	RemoteDevice		: FB_BACnet_RemoteDevice;
END_VAR
VAR_OUTPUT
	bReady				: BOOL;
	fControlledValue	: REAL;
	fPresentValue		: REAL;
	bOverridden			: BOOL;
	bOutOfService		: BOOL;
	bFault				: BOOL;
	bInAlarm			: BOOL;
	bError				: BOOL;
	nErrorId			: UINT;
END_VAR
VAR
	_PresentValue AT%I*: REAL; 				(* ~(BACnet_PresentValue 				: 		: )
												(BACnet_ObjectType					: LOOP	: )
			                                	(BACnet_RemoteCycletimeRead 		: 1000	: )
												(BACnet_RemoteFlagsRead        		: 1     : )
                                   				(BACnet_RemoteResubscriptionInterval: 240 	: )
		                                		(BACnet_RemoteCycleTimeWrite   		: 1000	: )
		                                		(BACnet_RemoteFlagsWrite       		: 1		: )	*)
	_ControlledVariableValue AT%I*: REAL; 	(* ~(BACnet_ControlledVariableValue 	:		: )	*)
	_StatusFlags AT%I*: WORD; 				(* ~(BACnet_StatusFlags 				:		: )	*)
	_StatusFlagsBits : ST_BACnet_StatusFlags;
	_nUpdateCount : UDINT := 0;
END_VAR
(* update client device *)
IF RemoteDevice._nUpdateCount = _nUpdateCount THEN
	RemoteDevice();
END_IF
(* remind current number of update counter *)
_nUpdateCount := RemoteDevice._nUpdateCount;

IF NOT RemoteDevice.bOperational THEN
	nErrorId := BACnet_ERR_OPERATIONAL;
	bReady := FALSE;

ELSIF _StatusFlags >= 4 THEN
	(* clear error flag *)
	nErrorId := BACnet_ERR_NO_ERROR;
	(* ready state *)
	bReady := TRUE;

	(* present value *)
	fPresentValue := _PresentValue;
	fControlledValue := _ControlledVariableValue;

	(* build bit states *)
	_StatusFlagsBits := F_BACnet_StatusFlags(_StatusFlags);

	(* copy states to output *)
	bOverridden := _StatusFlagsBits.overridden;
	bOutOfService := _StatusFlagsBits.out_of_service;
	bFault := _StatusFlagsBits.fault;
	bInAlarm := _StatusFlagsBits.in_alarm;
ELSE
	(* server device not ready, reset local ready also *)
	bReady := FALSE;
	(* and set error ID *)
	nErrorId := BACnet_ERR_WRONG_MAPPING;
END_IF

(* set error flag *)
bError := (nErrorId <> BACnet_ERR_NO_ERROR);
END_FUNCTION_BLOCK

(* POU FB_BACnet_RemoteLoop_EX, ST *)
FUNCTION_BLOCK FB_BACnet_RemoteLoop_EX
VAR_IN_OUT
	RemoteDevice		: FB_BACnet_RemoteDevice;
END_VAR
VAR_OUTPUT
	bReady				: BOOL;
	fControlledValue	: REAL;
	fPresentValue		: REAL;
	bOverridden			: BOOL;
	bOutOfService		: BOOL;
	bFault				: BOOL;
	bInAlarm			: BOOL;
	bOpenLoop			: BOOL;
	bOtherFault			: BOOL;
	eEventState			: E_BACNETEVENTSTATE;
	tObjectID			: T_BACnet_ObjectIdentifier := 16#FFFFFFFF;
	bError				: BOOL;
	nErrorId			: UINT;
END_VAR
VAR
	_PresentValue AT%I*: REAL; 			(* ~(BACnet_PresentValue 				: LP	: )
			                               	(BACnet_RemoteCycletimeRead 		: 1000	: )
											(BACnet_RemoteFlagsRead        		: 1     : )
                                   			(BACnet_RemoteResubscriptionInterval: 240 	: )
		                                	(BACnet_RemoteCycleTimeWrite   		: 1000	: )
		                                	(BACnet_RemoteFlagsWrite       		: 1		: )	*)
	_ControlledVariableValue AT%I*: REAL;(* ~(BACnet_ControlledVariableValue 	:		: )	*)
	_ObjectId AT%I*: DWORD;				(* ~(BACnet_ObjectIdentifier			:		: LINK) *)
	_Reliability AT%I*: WORD; 			(* ~(BACnet_Reliability 				:		: )	*)
	_StatusFlags AT%I*: WORD; 			(* ~(BACnet_StatusFlags 				:		: )	*)
	_EventState AT%I*: WORD;			(* ~(BACnet_EventState					:		: )	*)
	_nUpdateCount : UDINT := 0;
	_StatusFlagsBits : ST_BACnet_StatusFlags;
END_VAR
(* update client device *)
IF RemoteDevice._nUpdateCount = _nUpdateCount THEN
	RemoteDevice();
END_IF
(* remind current number of update counter *)
_nUpdateCount := RemoteDevice._nUpdateCount;

IF NOT RemoteDevice.bOperational THEN
	nErrorId := BACnet_ERR_OPERATIONAL;
	bReady := FALSE;

ELSIF (F_BACnet_GetObjType(_ObjectId) <> BACnetObjectType_Loop) THEN
	(* wrong mapping / invalid object ID *)
	IF _ObjectId = 0 THEN
		nErrorId := BACnet_ERR_WRONG_MAPPING;
	ELSE
		nErrorId := BACnet_ERR_INVALID_OBJECTID;
	END_IF
	bReady := FALSE;
	tObjectID := 16#FFFFFFFF;

ELSIF _StatusFlags >= 4 THEN
	(* clear error flag *)
	nErrorId := BACnet_ERR_NO_ERROR;
	(* ready state *)
	bReady := TRUE;

	(* present value *)
	fPresentValue := _PresentValue;
	fControlledValue := _ControlledVariableValue;

	(* build bit states *)
	_StatusFlagsBits := F_BACnet_StatusFlags(_StatusFlags);

	(* copy states to output *)
	bOverridden := _StatusFlagsBits.overridden;
	bOutOfService := _StatusFlagsBits.out_of_service;
	bFault := _StatusFlagsBits.fault;
	bInAlarm := _StatusFlagsBits.in_alarm;
	bOpenLoop := (_Reliability = BACnetReliability_open_loop);
	bOtherFault := (_Reliability = BACnetReliability_unreliable_other);
	eEventState := _EventState;
	tObjectID := _ObjectId;
ELSE
	(* server device not ready, reset local ready also *)
	bReady := FALSE;
	(* and set error ID *)
	nErrorId := BACnet_ERR_WRONG_MAPPING;
END_IF

(* set error flag *)
bError := (nErrorId <> BACnet_ERR_NO_ERROR);
END_FUNCTION_BLOCK

(* POU FB_BACnet_RemoteMultiStateInput, ST *)
FUNCTION_BLOCK FB_BACnet_RemoteMultiStateInput
VAR_IN_OUT
	RemoteDevice		: FB_BACnet_RemoteDevice;
END_VAR
VAR_OUTPUT
	bReady				: BOOL;
	nPresentValue		: UDINT;
	bOverridden			: BOOL;
	bOutOfService		: BOOL;
	bFault				: BOOL;
	bInAlarm			: BOOL;
	bError				: BOOL;
	nErrorId			: UINT;
END_VAR
VAR
	_PresentValue AT%I*: UDINT; 	(* ~(BACnet_PresentValue 				:		: )
								   		(BACnet_ObjectType 					: MI	: )
										(BACnet_RemoteCycletimeRead 		: 1000	: )
										(BACnet_RemoteFlagsRead        		: 1		: )
										(BACnet_RemoteResubscriptionInterval: 240	: )
                                		(BACnet_RemoteCycleTimeWrite   		: 1000	: )
                                		(BACnet_RemoteFlagsWrite       		: 1		: )	*)
	_StatusFlags AT%I*: WORD; 		(* ~(BACnet_StatusFlags 				:		: )	*)
	_StatusFlagsBits : ST_BACnet_StatusFlags;
	_nUpdateCount : UDINT := 0;
END_VAR
(* update client device *)
IF RemoteDevice._nUpdateCount = _nUpdateCount THEN
	RemoteDevice();
END_IF
(* remind current number of update counter *)
_nUpdateCount := RemoteDevice._nUpdateCount;

IF NOT RemoteDevice.bOperational THEN
	nErrorId := BACnet_ERR_OPERATIONAL;
	bReady := FALSE;

ELSIF _StatusFlags >= 4 THEN
	(* clear error flag *)
	nErrorId := BACnet_ERR_NO_ERROR;
	(* ready state *)
	bReady := TRUE;

	(* present value *)
	nPresentValue := _PresentValue;

	(* build bit states *)
	_StatusFlagsBits := F_BACnet_StatusFlags(_StatusFlags);

	(* copy states to output *)
	bOverridden := _StatusFlagsBits.overridden;
	bOutOfService := _StatusFlagsBits.out_of_service;
	bFault := _StatusFlagsBits.fault;
	bInAlarm := _StatusFlagsBits.in_alarm;

ELSE
	(* server device not ready, reset local ready also *)
	bReady := FALSE;
	(* and set error ID *)
	nErrorId := BACnet_ERR_WRONG_MAPPING;
END_IF

(* set error flag *)
bError := (nErrorId <> BACnet_ERR_NO_ERROR);
END_FUNCTION_BLOCK

(* POU FB_BACnet_RemoteMultiStateInput_EX, ST *)
FUNCTION_BLOCK FB_BACnet_RemoteMultiStateInput_EX
VAR_IN_OUT
	RemoteDevice		: FB_BACnet_RemoteDevice;
END_VAR
VAR_OUTPUT
	bReady				: BOOL;
	nPresentValue		: UDINT;
	bOverridden			: BOOL;
	bOutOfService		: BOOL;
	bFault				: BOOL;
	bInAlarm			: BOOL;
	bOverRange			: BOOL;
	bUnderRange			: BOOL;
	bNoSensor			: BOOL;
	bOpenLoop			: BOOL;
	bShortedLoop		: BOOL;
	bMultiStateFault	: BOOL;
	bOtherFault			: BOOL;
	eEventState			: E_BACNETEVENTSTATE;
	nNbrOfStates		: UDINT;
	tObjectID			: T_BACnet_ObjectIdentifier := 16#FFFFFFFF;
	bError				: BOOL;
	nErrorId			: UINT;
END_VAR
VAR
	_PresentValue AT%I*: UDINT; 		(* ~(BACnet_PresentValue 				:		: )
								   			(BACnet_ObjectType 					: MI	: )
											(BACnet_RemoteCycletimeRead 		: 1000	: )
											(BACnet_RemoteFlagsRead        		: 1		: )
											(BACnet_RemoteResubscriptionInterval: 240	: )
                                			(BACnet_RemoteCycleTimeWrite   		: 1000	: )
                                			(BACnet_RemoteFlagsWrite       		: 1		: )	*)
	_NumberOfStates AT%I*: UDINT;		(* ~(BACnet_NumberOfStates				:		: )	*)
	_ObjectId AT%I*: DWORD;				(* ~(BACnet_ObjectIdentifier			:		: LINK) *)
	_StatusFlags AT%I*: WORD; 			(* ~(BACnet_StatusFlags 				:		: )	*)
	_Reliability AT%I*: WORD; 			(* ~(BACnet_Reliability 				:		: )	*)
	_EventState AT%I*: WORD; 			(* ~(BACnet_EventState 					:		: )	*)
	_nUpdateCount : UDINT := 0;
	_StatusFlagsBits : ST_BACnet_StatusFlags;
END_VAR
(* update client device *)
IF RemoteDevice._nUpdateCount = _nUpdateCount THEN
	RemoteDevice();
END_IF
(* remind current number of update counter *)
_nUpdateCount := RemoteDevice._nUpdateCount;

IF NOT RemoteDevice.bOperational THEN
	nErrorId := BACnet_ERR_OPERATIONAL;
	bReady := FALSE;

ELSIF (F_BACnet_GetObjType(_ObjectId) <> BACnetObjectType_MultiStateInput) THEN
	(* wrong mapping / invalid object ID *)
	IF _ObjectId = 0 THEN
		nErrorId := BACnet_ERR_WRONG_MAPPING;
	ELSE
		nErrorId := BACnet_ERR_INVALID_OBJECTID;
	END_IF
	bReady := FALSE;
	tObjectID := 16#FFFFFFFF;

ELSIF _StatusFlags >= 4 THEN
	(* clear error flag *)
	nErrorId := BACnet_ERR_NO_ERROR;
	(* ready state *)
	bReady := TRUE;

	(* present value *)
	nPresentValue := _PresentValue;

	(* build bit states *)
	_StatusFlagsBits := F_BACnet_StatusFlags(_StatusFlags);

	(* copy states to output *)
	bOverridden := _StatusFlagsBits.overridden;
	bOutOfService := _StatusFlagsBits.out_of_service;
	bFault := _StatusFlagsBits.fault;
	bInAlarm := _StatusFlagsBits.in_alarm;
	bOverRange := (_Reliability = BACnetReliability_over_range);
	bUnderRange := (_Reliability = BACnetReliability_under_range);
	bNoSensor := (_Reliability = BACnetReliability_no_sensor);
	bOpenLoop := (_Reliability = BACnetReliability_open_loop);
	bShortedLoop := (_Reliability = BACnetReliability_shorted_loop);
	bMultiStateFault := (_Reliability = BACnetReliability_multi_state_fault);
	bOtherFault := (_Reliability = BACnetReliability_unreliable_other);
	nNbrOfStates := _NumberOfStates;
	eEventState := _EventState;
	tObjectID := _ObjectId;

ELSE
	(* server device not ready, reset local ready also *)
	bReady := FALSE;
	(* and set error ID *)
	nErrorId := BACnet_ERR_WRONG_MAPPING;
END_IF

(* set error flag *)
bError := (nErrorId <> BACnet_ERR_NO_ERROR);
END_FUNCTION_BLOCK

(* POU FB_BACnet_RemoteMultiStateOutput, ST *)
FUNCTION_BLOCK FB_BACnet_RemoteMultiStateOutput
VAR_IN_OUT
	RemoteDevice		: FB_BACnet_RemoteDevice;
END_VAR
VAR_OUTPUT
	bReady				: BOOL;
	nPresentValue		: UDINT;
	bOverridden			: BOOL;
	bOutOfService		: BOOL;
	bFault				: BOOL;
	bInAlarm			: BOOL;
	nNbrOfStates		: UDINT;
	bError				: BOOL;
	nErrorId			: UINT;
END_VAR
VAR
	_PresentValue AT%I*: UDINT; 			(* ~(BACnet_PresentValue 				:		: )
								   				(BACnet_ObjectType					: MO	: )
												(BACnet_RemoteCycletimeRead 		: 1000	: )
												(BACnet_RemoteFlagsRead        		: 1		: )
												(BACnet_RemoteResubscriptionInterval: 240	: )
		                                		(BACnet_RemoteCycleTimeWrite   		: 1000	: )
		                                		(BACnet_RemoteFlagsWrite       		: 1		: )	*)
	_NumberOfStates AT%I*: UDINT;			(* ~(BACnet_NumberOfStates				:		: )	*)
	_StatusFlags AT%I*: WORD; 				(* ~(BACnet_StatusFlags					:		: )	*)
	_StatusFlagsBits : ST_BACnet_StatusFlags;
	_nUpdateCount : UDINT := 0;
END_VAR
(* update client device *)
IF RemoteDevice._nUpdateCount = _nUpdateCount THEN
	RemoteDevice();
END_IF
(* remind current number of update counter *)
_nUpdateCount := RemoteDevice._nUpdateCount;

IF RemoteDevice.bFirstCycle THEN
	(* first call of the server device since reboot/reset *)
	bReady := FALSE;

ELSIF NOT RemoteDevice.bOperational THEN
	nErrorId := BACnet_ERR_OPERATIONAL;
	bReady := FALSE;

ELSIF _StatusFlags >= 4 THEN
	(* clear error flag *)
	nErrorId := BACnet_ERR_NO_ERROR;
	(* ready state *)
	bReady := TRUE;

	(* present value *)
	nPresentValue := _PresentValue;

	(* build bit states *)
	_StatusFlagsBits := F_BACnet_StatusFlags(_StatusFlags);

	(* copy states to output *)
	bOverridden := _StatusFlagsBits.overridden;
	bOutOfService := _StatusFlagsBits.out_of_service;
	bFault := _StatusFlagsBits.fault;
	bInAlarm := _StatusFlagsBits.in_alarm;

	(* number of states *)
	nNbrOfStates := _NumberOfStates;

ELSE
	(* server device not ready, reset local ready also *)
	bReady := FALSE;
	(* and set error ID *)
	nErrorId := BACnet_ERR_WRONG_MAPPING;
END_IF

(* set error flag *)
bError := (nErrorId <> BACnet_ERR_NO_ERROR);
END_FUNCTION_BLOCK

(* POU FB_BACnet_RemoteMultiStateOutput_EX, ST *)
FUNCTION_BLOCK FB_BACnet_RemoteMultiStateOutput_EX
VAR_INPUT
	bEnablePV			: BOOL; (* enable present value with priority x in priority array, FALSE = priority x disable *)
	bNullPV				: BOOL; (* clear priority entry *)
	nPV					: UDINT; (* number for priority x, when input bEnablePV is TRUE *)
END_VAR
VAR_IN_OUT
	RemoteDevice		: FB_BACnet_RemoteDevice;
END_VAR
VAR_OUTPUT
	bReady				: BOOL;
	nPresentValue		: UDINT;
	bOverridden			: BOOL;
	bOutOfService		: BOOL;
	bFault				: BOOL;
	bInAlarm			: BOOL;
	bNoOutput			: BOOL;
	bOpenLoop			: BOOL;
	bShortedLoop		: BOOL;
	bOtherFault			: BOOL;
	eEventState			: E_BACNETEVENTSTATE;
	nActivePrio			: UINT;
	nNbrOfStates		: UDINT;
	tObjectID			: T_BACnet_ObjectIdentifier := 16#FFFFFFFF;
	bError				: BOOL;
	nErrorId			: UINT;
END_VAR
VAR
	_PresentValue AT%I*: UDINT; 		(* ~(BACnet_PresentValue 				:		: )
								   			(BACnet_ObjectType					: MO	: )
											(BACnet_RemoteCycletimeRead 		: 1000	: )
											(BACnet_RemoteFlagsRead        		: 1		: )
											(BACnet_RemoteResubscriptionInterval: 240	: )
		                                	(BACnet_RemoteCycleTimeWrite   		: 1000	: )
		                                	(BACnet_RemoteFlagsWrite       		: 1		: )	*)
	_NumberOfStates AT%I*: UDINT;		(* ~(BACnet_NumberOfStates				:		: )	*)
	_ActivePriority AT%I*: UDINT; 		(* ~(BACnet_ActivePriority 				:		: )	*)
	_ObjectId AT%I*: DWORD;				(* ~(BACnet_ObjectIdentifier			:		: LINK) *)
	_StatusFlags AT%I*: WORD; 			(* ~(BACnet_StatusFlags					:		: )	*)
	_Reliability AT%I*: WORD; 			(* ~(BACnet_Reliability					:		: )	*)
	_EventState AT%I*: WORD;			(* ~(BACnet_EventState					:		: )	*)
    _PresentValue_Priority12 AT%Q*: UDINT;(* ~(BACnet_PresentValue_Priority12	:		: )	*)
	_nUpdateCount : UDINT := 0;
	_StatusFlagsBits : ST_BACnet_StatusFlags;
END_VAR
(* update client device *)
IF RemoteDevice._nUpdateCount = _nUpdateCount THEN
	RemoteDevice();
END_IF
(* remind current number of update counter *)
_nUpdateCount := RemoteDevice._nUpdateCount;

IF RemoteDevice.bFirstCycle THEN
	(* first call of the server device since reboot/reset *)
	bReady := FALSE;
	_PresentValue_Priority12 := 16#FFFFFFFF;
ELSIF NOT RemoteDevice.bOperational THEN
	nErrorId := BACnet_ERR_OPERATIONAL;
	bReady := FALSE;

ELSIF (F_BACnet_GetObjType(_ObjectId) <> BACnetObjectType_MultiStateOutput) THEN
	(* wrong mapping / invalid object ID *)
	IF _ObjectId = 0 THEN
		nErrorId := BACnet_ERR_WRONG_MAPPING;
	ELSE
		nErrorId := BACnet_ERR_INVALID_OBJECTID;
	END_IF
	bReady := FALSE;
	tObjectID := 16#FFFFFFFF;

ELSIF _StatusFlags >= 4 THEN
	(* clear error flag *)
	nErrorId := BACnet_ERR_NO_ERROR;
	(* ready state *)
	bReady := TRUE;

	(* write into priority array *)
	_PresentValue_Priority12 := F_BACnet_MultiStatePV(bEnablePV, bNullPV, nPV);

	(* present value *)
	nPresentValue := _PresentValue;

	(* build bit states *)
	_StatusFlagsBits := F_BACnet_StatusFlags(_StatusFlags);

	(* copy states to output *)
	bOverridden := _StatusFlagsBits.overridden;
	bOutOfService := _StatusFlagsBits.out_of_service;
	bFault := _StatusFlagsBits.fault;
	bInAlarm := _StatusFlagsBits.in_alarm;
	bNoOutput := (_Reliability = BACnetReliability_no_output);
	bOpenLoop := (_Reliability = BACnetReliability_open_loop);
	bShortedLoop := (_Reliability = BACnetReliability_shorted_loop);
	bOtherFault := (_Reliability = BACnetReliability_unreliable_other);
	eEventState := _EventState;
	tObjectID := _ObjectId;

	(* copy active priority *)
	nActivePrio := UDINT_TO_UINT(_ActivePriority);

	(* number of states *)
	nNbrOfStates := _NumberOfStates;

ELSE
	(* server device not ready, reset local ready also *)
	bReady := FALSE;
	(* and set error ID *)
	nErrorId := BACnet_ERR_WRONG_MAPPING;
END_IF

(* set error flag *)
bError := (nErrorId <> BACnet_ERR_NO_ERROR);
END_FUNCTION_BLOCK

(* POU FB_BACnet_RemoteMultiStateOutput_WR, ST *)
FUNCTION_BLOCK FB_BACnet_RemoteMultiStateOutput_WR
VAR_INPUT
	bEnablePV			: BOOL; (* enable present value with priority x in priority array, FALSE = priority x disable *)
	bNullPV				: BOOL; (* clear priority entry *)
	nPV					: UDINT; (* number for priority x, when input bEnablePV is TRUE *)
END_VAR
VAR_IN_OUT
	RemoteDevice		: FB_BACnet_RemoteDevice;
END_VAR
VAR_OUTPUT
	bReady				: BOOL;
	nPresentValue		: UDINT;
	bOverridden			: BOOL;
	bOutOfService		: BOOL;
	bFault				: BOOL;
	bInAlarm			: BOOL;
	nNbrOfStates		: UDINT;
	bError				: BOOL;
	nErrorId			: UINT;
END_VAR
VAR
	_PresentValue AT%I*: UDINT; 			(* ~(BACnet_PresentValue 				:		: )
								   				(BACnet_ObjectType					: MO	: )
												(BACnet_RemoteCycletimeRead 		: 1000	: )
												(BACnet_RemoteFlagsRead        		: 1		: )
												(BACnet_RemoteResubscriptionInterval: 240	: )
		                                		(BACnet_RemoteCycleTimeWrite   		: 1000	: )
		                                		(BACnet_RemoteFlagsWrite       		: 1		: )	*)
	_NumberOfStates AT%I*: UDINT;			(* ~(BACnet_NumberOfStates				:		: )	*)
	_StatusFlags AT%I*: WORD; 				(* ~(BACnet_StatusFlags					:		: )	*)
    _PresentValue_Priority12 AT%Q*: UDINT;	(* ~(BACnet_PresentValue_Priority12		:		: )	*)
	_StatusFlagsBits : ST_BACnet_StatusFlags;
	_nUpdateCount : UDINT := 0;
END_VAR
(* update client device *)
IF RemoteDevice._nUpdateCount = _nUpdateCount THEN
	RemoteDevice();
END_IF
(* remind current number of update counter *)
_nUpdateCount := RemoteDevice._nUpdateCount;

IF RemoteDevice.bFirstCycle THEN
	(* first call of the server device since reboot/reset *)
	bReady := FALSE;
	_PresentValue_Priority12 := 16#FFFFFFFF;
ELSIF NOT RemoteDevice.bOperational THEN
	nErrorId := BACnet_ERR_OPERATIONAL;
	bReady := FALSE;

ELSIF _StatusFlags >= 4 THEN
	(* clear error flag *)
	nErrorId := BACnet_ERR_NO_ERROR;
	(* ready state *)
	bReady := TRUE;

	(* write into priority array *)
	_PresentValue_Priority12 := F_BACnet_MultiStatePV(bEnablePV, bNullPV, nPV);

	(* present value *)
	nPresentValue := _PresentValue;

	(* build bit states *)
	_StatusFlagsBits := F_BACnet_StatusFlags(_StatusFlags);

	(* copy states to output *)
	bOverridden := _StatusFlagsBits.overridden;
	bOutOfService := _StatusFlagsBits.out_of_service;
	bFault := _StatusFlagsBits.fault;
	bInAlarm := _StatusFlagsBits.in_alarm;

	(* number of states *)
	nNbrOfStates := _NumberOfStates;

ELSE
	(* server device not ready, reset local ready also *)
	bReady := FALSE;
	(* and set error ID *)
	nErrorId := BACnet_ERR_WRONG_MAPPING;
END_IF

(* set error flag *)
bError := (nErrorId <> BACnet_ERR_NO_ERROR);
END_FUNCTION_BLOCK

(* POU FB_BACnet_RemoteMultiStateValue, ST *)
FUNCTION_BLOCK FB_BACnet_RemoteMultiStateValue
VAR_IN_OUT
	RemoteDevice		: FB_BACnet_RemoteDevice;
END_VAR
VAR_OUTPUT
	bReady				: BOOL;
	nPresentValue		: UDINT;
	bOverridden			: BOOL;
	bOutOfService		: BOOL;
	bFault				: BOOL;
	bInAlarm			: BOOL;
	nNbrOfStates		: UDINT;
	bError				: BOOL;
	nErrorId			: UINT;
END_VAR
VAR
	_PresentValue AT%I*: UDINT; 			(* ~(BACnet_PresentValue 				:		: )
								   				(BACnet_ObjectType 					: MV	: )
												(BACnet_RemoteCycletimeRead 		: 1000	: )
												(BACnet_RemoteFlagsRead        		: 1		: )
												(BACnet_RemoteResubscriptionInterval: 240	: )
		                                		(BACnet_RemoteCycleTimeWrite   		: 1000	: )
		                                		(BACnet_RemoteFlagsWrite       		: 1		: )	*)
	_NumberOfStates AT%I*: UDINT;			(* ~(BACnet_NumberOfStates				:		: )	*)
	_StatusFlags AT%I*: WORD; 				(* ~(BACnet_StatusFlags 				:		: )	*)
	_StatusFlagsBits : ST_BACnet_StatusFlags;
	_nUpdateCount : UDINT := 0;
END_VAR
(* update client device *)
IF RemoteDevice._nUpdateCount = _nUpdateCount THEN
	RemoteDevice();
END_IF
(* remind current number of update counter *)
_nUpdateCount := RemoteDevice._nUpdateCount;

IF RemoteDevice.bFirstCycle THEN
	(* first call of the server device since reboot/reset *)
	bReady := FALSE;

ELSIF NOT RemoteDevice.bOperational THEN
	nErrorId := BACnet_ERR_OPERATIONAL;
	bReady := FALSE;

ELSIF _StatusFlags >= 4 THEN
	(* clear error flag *)
	nErrorId := BACnet_ERR_NO_ERROR;
	(* ready state *)
	bReady := TRUE;

	(* present value *)
	nPresentValue := _PresentValue;

	(* build bit states *)
	_StatusFlagsBits := F_BACnet_StatusFlags(_StatusFlags);

	(* copy states to output *)
	bOverridden := _StatusFlagsBits.overridden;
	bOutOfService := _StatusFlagsBits.out_of_service;
	bFault := _StatusFlagsBits.fault;
	bInAlarm := _StatusFlagsBits.in_alarm;

	(* number of states *)
	nNbrOfStates := _NumberOfStates;

ELSE
	(* server device not ready, reset local ready also *)
	bReady := FALSE;
	(* and set error ID *)
	nErrorId := BACnet_ERR_WRONG_MAPPING;
END_IF

(* set error flag *)
bError := (nErrorId <> BACnet_ERR_NO_ERROR);
END_FUNCTION_BLOCK

(* POU FB_BACnet_RemoteMultiStateValue_EX, ST *)
FUNCTION_BLOCK FB_BACnet_RemoteMultiStateValue_EX
VAR_INPUT
	bEnablePV			: BOOL; (* enable present value with priority x in priority array, FALSE = priority x disable *)
	bNullPV				: BOOL; (* clear priority entry *)
	nPV					: UDINT; (* number for priority x, when input bEnablePV is TRUE *)
END_VAR
VAR_IN_OUT
	RemoteDevice		: FB_BACnet_RemoteDevice;
END_VAR
VAR_OUTPUT
	bReady				: BOOL;
	nPresentValue		: UDINT;
	bOverridden			: BOOL;
	bOutOfService		: BOOL;
	bFault				: BOOL;
	bInAlarm			: BOOL;
	bMultiStateFault	: BOOL;
	bOtherFault			: BOOL;
	eEventState			: E_BACNETEVENTSTATE;
	nNbrOfStates		: UDINT;
	tObjectID			: T_BACnet_ObjectIdentifier := 16#FFFFFFFF;
	bError				: BOOL;
	nErrorId			: UINT;
END_VAR
VAR
	_PresentValue AT%I*: UDINT; 		(* ~(BACnet_PresentValue 				:		: )
											(BACnet_ObjectType 					: MV	: )
											(BACnet_RemoteCycletimeRead 		: 1000	: )
											(BACnet_RemoteFlagsRead        		: 1		: )
											(BACnet_RemoteResubscriptionInterval: 240	: )
											(BACnet_RemoteCycleTimeWrite   		: 1000	: )
											(BACnet_RemoteFlagsWrite       		: 1		: )	*)
	_NumberOfStates AT%I*: UDINT;		(* ~(BACnet_NumberOfStates				:		: )	*)
	_EventState AT%I*: WORD;			(* ~(BACnet_EventState					:		: )	*)
	_ObjectId AT%I*: DWORD;				(* ~(BACnet_ObjectIdentifier			:		: LINK) *)
	_StatusFlags AT%I*: WORD;			(* ~(BACnet_StatusFlags 				:		: )	*)
	_Reliability AT%I*: WORD;			(* ~(BACnet_Reliability 				:		: )	*)
    _PresentValue_Priority12 AT%Q*: UDINT;(* ~(BACnet_PresentValue_Priority12	:		: )	*)
	_nUpdateCount : UDINT := 0;
	_StatusFlagsBits : ST_BACnet_StatusFlags;
END_VAR
(* update client device *)
IF RemoteDevice._nUpdateCount = _nUpdateCount THEN
	RemoteDevice();
END_IF
(* remind current number of update counter *)
_nUpdateCount := RemoteDevice._nUpdateCount;

IF RemoteDevice.bFirstCycle THEN
	(* first call of the server device since reboot/reset *)
	bReady := FALSE;
	_PresentValue_Priority12 := 16#FFFFFFFF;
ELSIF NOT RemoteDevice.bOperational THEN
	nErrorId := BACnet_ERR_OPERATIONAL;
	bReady := FALSE;

ELSIF (F_BACnet_GetObjType(_ObjectId) <> BACnetObjectType_MultiStateValue) THEN
	(* wrong mapping / invalid object ID *)
	IF _ObjectId = 0 THEN
		nErrorId := BACnet_ERR_WRONG_MAPPING;
	ELSE
		nErrorId := BACnet_ERR_INVALID_OBJECTID;
	END_IF
	bReady := FALSE;
	tObjectID := 16#FFFFFFFF;

ELSIF _StatusFlags >= 4 THEN
	(* clear error flag *)
	nErrorId := BACnet_ERR_NO_ERROR;
	(* ready state *)
	bReady := TRUE;

	(* write into priority array *)
	_PresentValue_Priority12 := F_BACnet_MultiStatePV(bEnablePV, bNullPV, nPV);

	(* present value *)
	nPresentValue := _PresentValue;

	(* build bit states *)
	_StatusFlagsBits := F_BACnet_StatusFlags(_StatusFlags);

	(* copy states to output *)
	bOverridden := _StatusFlagsBits.overridden;
	bOutOfService := _StatusFlagsBits.out_of_service;
	bFault := _StatusFlagsBits.fault;
	bInAlarm := _StatusFlagsBits.in_alarm;
	bMultiStateFault := (_Reliability = BACnetReliability_multi_state_fault);
	bOtherFault := (_Reliability = BACnetReliability_unreliable_other);
	eEventState := _EventState;
	tObjectID := _ObjectId;

	(* number of states *)
	nNbrOfStates := _NumberOfStates;

ELSE
	(* server device not ready, reset local ready also *)
	bReady := FALSE;
	(* and set error ID *)
	nErrorId := BACnet_ERR_WRONG_MAPPING;
END_IF

(* set error flag *)
bError := (nErrorId <> BACnet_ERR_NO_ERROR);
END_FUNCTION_BLOCK

(* POU FB_BACnet_RemoteMultiStateValue_WR, ST *)
FUNCTION_BLOCK FB_BACnet_RemoteMultiStateValue_WR
VAR_INPUT
	bEnablePV			: BOOL; (* enable present value with priority x in priority array, FALSE = priority x disable *)
	bNullPV				: BOOL; (* clear priority entry *)
	nPV					: UDINT; (* number for priority x, when input bEnablePV is TRUE *)
END_VAR
VAR_IN_OUT
	RemoteDevice		: FB_BACnet_RemoteDevice;
END_VAR
VAR_OUTPUT
	bReady				: BOOL;
	nPresentValue		: UDINT;
	bOverridden			: BOOL;
	bOutOfService		: BOOL;
	bFault				: BOOL;
	bInAlarm			: BOOL;
	nNbrOfStates		: UDINT;
	bError				: BOOL;
	nErrorId			: UINT;
END_VAR
VAR
	_PresentValue AT%I*: UDINT; 			(* ~(BACnet_PresentValue 				:		: )
								   				(BACnet_ObjectType 					: MV	: )
												(BACnet_RemoteCycletimeRead 		: 1000	: )
												(BACnet_RemoteFlagsRead        		: 1		: )
												(BACnet_RemoteResubscriptionInterval: 240	: )
		                                		(BACnet_RemoteCycleTimeWrite   		: 1000	: )
		                                		(BACnet_RemoteFlagsWrite       		: 1		: )	*)
	_NumberOfStates AT%I*: UDINT;			(* ~(BACnet_NumberOfStates				:		: )	*)
	_StatusFlags AT%I*: WORD; 				(* ~(BACnet_StatusFlags 				:		: )	*)
    _PresentValue_Priority12 AT%Q*: UDINT;	(* ~(BACnet_PresentValue_Priority12		:		: )	*)
	_StatusFlagsBits : ST_BACnet_StatusFlags;
	_nUpdateCount : UDINT := 0;
END_VAR
(* update client device *)
IF RemoteDevice._nUpdateCount = _nUpdateCount THEN
	RemoteDevice();
END_IF
(* remind current number of update counter *)
_nUpdateCount := RemoteDevice._nUpdateCount;

IF RemoteDevice.bFirstCycle THEN
	(* first call of the server device since reboot/reset *)
	bReady := FALSE;
	_PresentValue_Priority12 := 16#FFFFFFFF;
ELSIF NOT RemoteDevice.bOperational THEN
	nErrorId := BACnet_ERR_OPERATIONAL;
	bReady := FALSE;

ELSIF _StatusFlags >= 4 THEN
	(* clear error flag *)
	nErrorId := BACnet_ERR_NO_ERROR;
	(* ready state *)
	bReady := TRUE;

	(* write into priority array *)
	_PresentValue_Priority12 := F_BACnet_MultiStatePV(bEnablePV, bNullPV, nPV);

	(* present value *)
	nPresentValue := _PresentValue;

	(* build bit states *)
	_StatusFlagsBits := F_BACnet_StatusFlags(_StatusFlags);

	(* copy states to output *)
	bOverridden := _StatusFlagsBits.overridden;
	bOutOfService := _StatusFlagsBits.out_of_service;
	bFault := _StatusFlagsBits.fault;
	bInAlarm := _StatusFlagsBits.in_alarm;

	(* number of states *)
	nNbrOfStates := _NumberOfStates;

ELSE
	(* server device not ready, reset local ready also *)
	bReady := FALSE;
	(* and set error ID *)
	nErrorId := BACnet_ERR_WRONG_MAPPING;
END_IF

(* set error flag *)
bError := (nErrorId <> BACnet_ERR_NO_ERROR);
END_FUNCTION_BLOCK

(* POU FB_BACnet_RemoteNotificationClass, ST *)
FUNCTION_BLOCK FB_BACnet_RemoteNotificationClass
VAR_IN_OUT
	RemoteDevice		: FB_BACnet_RemoteDevice;
END_VAR
VAR_OUTPUT
	bReady				: BOOL;
	bError				: BOOL;
	nErrorId			: UINT;
END_VAR
VAR
	_ObjectType : E_BACNETOBJECTTYPE; (* ~(BACNET_OBJECTTYPE :NC:)  *)
	_nUpdateCount : UDINT := 0;
END_VAR
_ObjectType := BACnetObjectType_NotificationClass;
(* update client device *)
IF RemoteDevice._nUpdateCount = _nUpdateCount THEN
	RemoteDevice();
END_IF
(* remind current number of update counter *)
_nUpdateCount := RemoteDevice._nUpdateCount;

IF RemoteDevice.bOperational THEN
	(* clear error flag *)
	nErrorId := BACnet_ERR_NO_ERROR;
	(* ready state *)
	bReady := TRUE;
ELSE
	(* server device not ready, reset local ready also *)
	bReady := FALSE;
	(* and set error ID *)
	nErrorId := BACnet_ERR_OPERATIONAL;
END_IF

(* set error flag *)
bError := (nErrorId <> BACnet_ERR_NO_ERROR);
END_FUNCTION_BLOCK

(* POU FB_BACnet_RemoteNotificationClass_EX, ST *)
FUNCTION_BLOCK FB_BACnet_RemoteNotificationClass_EX
VAR_IN_OUT
	RemoteDevice		: FB_BACnet_RemoteDevice;
END_VAR
VAR_OUTPUT
	bReady				: BOOL;
	tObjectID			: T_BACnet_ObjectIdentifier := 16#FFFFFFFF;
	bError				: BOOL;
	nErrorId			: UINT;
END_VAR
VAR
	_ObjectId AT%I*: DWORD;				(* ~(BACnet_ObjectIdentifier	:		: LINK)
											(BACNET_OBJECTTYPE			: NC	: ) *)
	_nUpdateCount : UDINT := 0;
END_VAR
(* update client device *)
IF RemoteDevice._nUpdateCount = _nUpdateCount THEN
	RemoteDevice();
END_IF
(* remind current number of update counter *)
_nUpdateCount := RemoteDevice._nUpdateCount;

IF NOT RemoteDevice.bOperational THEN
	(* server device not ready, reset local ready also *)
	bReady := FALSE;
	(* and set error ID *)
	nErrorId := BACnet_ERR_OPERATIONAL;

ELSIF (F_BACnet_GetObjType(_ObjectId) <> BACnetObjectType_NotificationClass) THEN
	(* wrong mapping / invalid object ID *)
	IF _ObjectId = 0 THEN
		nErrorId := BACnet_ERR_WRONG_MAPPING;
	ELSE
		nErrorId := BACnet_ERR_INVALID_OBJECTID;
	END_IF
	bReady := FALSE;
	tObjectID := 16#FFFFFFFF;

ELSIF RemoteDevice.bOperational THEN
	(* clear error flag *)
	nErrorId := BACnet_ERR_NO_ERROR;
	(* ready state *)
	bReady := TRUE;
	tObjectID := _ObjectId;

END_IF

(* set error flag *)
bError := (nErrorId <> BACnet_ERR_NO_ERROR);
END_FUNCTION_BLOCK

